(* PLC project mtcs_common, Institute of Astronomy OntoManager 0.0.1 *)
(* stored: creationDateTime 2017-02-10T20:20:17.105900, modificationDateTime 2017-02-10T20:20:17.105900 *)

TYPE InitializationStates : (SHUTDOWN := 0, INITIALIZING := 1, INITIALIZING_FAILED := 2, INITIALIZED := 3, LOCKED := 4);
END_TYPE

TYPE OperatorStates : (NONE := 0, OBSERVER := 1, TECH := 2);
END_TYPE

TYPE OperatingStates : (AUTO := 0, MANUAL := 1);
END_TYPE

TYPE LimitSwitches : (POSITIVE_LIMIT_SWITCH := 0, NEGATIVE_LIMIT_SWITCH := 1);
END_TYPE

TYPE Units : (DEGREE := 0, RADIAN := 1, PERCENT := 2, RADIANS_PER_SECOND := 3, DEGREES_PER_SECOND := 4, MILLIMETERS_PER_SECOND := 5, REVOLUTIONS_PER_SECOND := 6, REVOLUTIONS_PER_MINUTE := 7, AMPS := 8, MILLIAMPS := 9, MILLIMETER := 10, MICROMETER := 11, DEGREES_CELSIUS := 12, KELVIN := 13, BAR := 14, PASCAL := 15, UNITLESS := 16, NEWTON := 17, DECANEWTON := 18, VOLT := 19, MILLIVOLT := 20, HERTZ := 21, G := 22, MILLIG := 23, NEWTONMETER := 24, ARCSECONDS := 25, ARCSECONDS_PER_SECOND := 26, RADIANS_PER_SQUARE_SECOND := 27, DEGREES_PER_SQUARE_SECOND := 28, ARCSECONDS_PER_SQUARE_SECOND := 29, METERS_PER_SECOND := 30, HECTOPASCAL := 31, SECONDS := 32, MINUTES := 33, MILLIMETERS_PER_HOUR := 34, HITS_PER_SQUARE_CENTIMETER := 35, HITS_PER_SQUARE_CENTIMETER_PER_HOUR := 36);
END_TYPE

TYPE RequestResults : (ACCEPTED := 0, REJECTED := 1);
END_TYPE

TYPE DriveOperatingModes : (OPERATING_MODE_NONE := 0, OPERATING_MODE_TORQUE_CONTROL := 1, OPERATING_MODE_VELOCITY_CONTROL := 2, OPERATING_MODE_POSITION_CONTROL := 3);
END_TYPE

TYPE DriveBrakeStates : (BRAKE_AUTOMATIC := 0, BRAKE_FORCE_LOCK := 1, BRAKE_FORCE_UNLOCK := 2);
END_TYPE

TYPE AX52XXDriveParts : STRUCT
  channelA : AX52XXDriveChannel;  (* Channel A *)
  channelB : AX52XXDriveChannel;  (* Channel B *)
END_STRUCT;
END_TYPE

TYPE BaseAxisProcesses : STRUCT
  moveAbsolute : McMoveAbsoluteProcess;  (* Move absolute *)
  moveRelative : McMoveRelativeProcess;  (* Move relative *)
  moveVelocity : McMoveVelocityProcess;  (* Move at a constant velocity *)
  reset : McProcess;  (* Reset any errors *)
  stop : McProcess;  (* Stop any movement *)
  stopParametrized : McStopProcess;  (* Stop any movement *)
  power : McPowerProcess;  (* Power on/off the axis *)
  gearIn : McProcess;  (* Couple to master axis *)
  gearOut : McProcess;  (* Decouple from master axis *)
  initialize : Process;  (* Start initializing the axis *)
  setPosition : McSetPositionProcess;  (* Set the axis position *)
  enableExtSetGen : McProcess;  (* Enable the external setpoint generator *)
  disableExtSetGen : McProcess;  (* Disable the external setpoint generator *)
  forceCalibration : McProcess;  (* Force the calibration (homing) flag to TRUE *)
  resetCalibration : McProcess;  (* Reset the calibration (homing) flag to FALSE *)
  readParameter : McReadParameter;  (* Read a numerical parameter *)
  readBoolParameter : McReadBoolParameter;  (* Read a boolean parameter *)
  writeParameter : McWriteParameter;  (* Write a numerical parameter *)
  writeBoolParameter : McWriteBoolParameter;  (* Write a boolean parameter *)
END_STRUCT;
END_TYPE

TYPE FaulhaberDriveProcesses : STRUCT
  write : SDOWriteProcess;  (* Write a number of bytes to the drive *)
  read : SDOReadProcess;  (* Read a number of bytes from the drive *)
  initialize : Process;  (* Initialize the drive according to the config *)
END_STRUCT;
END_TYPE

TYPE AX52XXDriveChannelProcesses : STRUCT
  read : SoEReadProcess;  (* Read a number of bytes from the drive *)
  write : SoEWriteProcess;  (* Write a number of bytes to the drive *)
  update : Process;  (* Update the actual values *)
  reset : SoEResetProcess;  (* Reset the drive channel *)
  acknowledgeSafetyError : Process;  (* Acknowledge the safety card error state *)
  setBrake : SetBrakeProcess;  (* Update the actual values *)
END_STRUCT;
END_TYPE

TYPE IncrementalEncoderProcesses : STRUCT
  enableCounterResetC : Process;  (* Enable the counter reset on the C pulse *)
  disableCounterResetC : Process;  (* Disable the counter reset on the C pulse *)
END_STRUCT;
END_TYPE

TYPE SimpleRelayProcesses : STRUCT
  setEnabled : SetEnabledProcess;  (* Set the relay enabled or disabled *)
END_STRUCT;
END_TYPE

TYPE ConfigManagerProcesses : STRUCT
  save : WriteXmlProcess;  (* Save the currently active config to disk *)
  load : ReadXmlProcess;  (* Load the config from disk *)
  activate : ActivateProcess;  (* Activate the loaded config *)
END_STRUCT;
END_TYPE

TYPE ModbusRTUBusProcesses : STRUCT
  readCoil : ModbusRTUBusReadCoilProcess;  (* Read coil *)
  writeCoil : ModbusRTUBusWriteCoilProcess;  (* Write coil *)
  readRegister : ModbusRTUBusReadRegisterProcess;  (* Read register *)
  writeRegister : ModbusRTUBusWriteRegisterProcess;  (* Write register *)
END_STRUCT;
END_TYPE

TYPE BaseProcessStatuses : STRUCT
  enabledStatus : EnabledStatus;  (* Is the process enabled or not? *)
  busyStatus : BusyStatus;  (* Is the process busy or not? *)
  healthStatus : HealthStatus;  (* Is the process in a healthy state or not? *)
  startedStatus : StartedStatus;  (* Is the process started or not? *)
END_STRUCT;
END_TYPE

TYPE ProcessStepStatuses : STRUCT
  enabledStatus : EnabledStatus;  (* Is the process step enabled or not? *)
END_STRUCT;
END_TYPE

TYPE BaseAxisStatuses : STRUCT
  busyStatus : BusyStatus;  (* Is the NcAxis in a busy state? *)
  healthStatus : HealthStatus;  (* Is the NcAxis in a healthy state? *)
  poweredStatus : PoweredStatus;  (* Is the NcAxis powered? *)
  extSetGenStatus : EnabledStatus;  (* Is the NcAxis its external setpoint generator enabled? *)
  motionStatus : MotionStatus;  (* Is the NcAxis moving forward or backward or standing still? *)
END_STRUCT;
END_TYPE

TYPE FaulhaberDriveStatuses : STRUCT
  busyStatus : BusyStatus;  (* Is the NcAxis in a busy state? *)
  healthStatus : HealthStatus;  (* Is the NcAxis in a healthy state? *)
END_STRUCT;
END_TYPE

TYPE AX52XXDriveChannelStatuses : STRUCT
  busyStatus : BusyStatus;  (* Is the drive in a busy state? *)
  healthStatus : HealthStatus;  (* Is the drive in a healthy state? *)
END_STRUCT;
END_TYPE

TYPE AX52XXDriveStatuses : STRUCT
  busyStatus : BusyStatus;  (* Is the drive in a busy state? *)
  healthStatus : HealthStatus;  (* Is the drive in a healthy state? *)
END_STRUCT;
END_TYPE

TYPE SSIEncoderStatuses : STRUCT
  healthStatus : HealthStatus;  (* Is the device in a healthy state? *)
END_STRUCT;
END_TYPE

TYPE IncrementalEncoderStatuses : STRUCT
  healthStatus : HealthStatus;  (* Is the device in a healthy state? *)
  busyStatus : BusyStatus;  (* Is the device in a busy state? *)
END_STRUCT;
END_TYPE

TYPE EtherCatDeviceStatuses : STRUCT
  healthStatus : HealthStatus;  (* Is the device in a healthy state? *)
END_STRUCT;
END_TYPE

TYPE CANopenBusStatuses : STRUCT
  healthStatus : HealthStatus;  (* Is the device in a healthy state? *)
END_STRUCT;
END_TYPE

TYPE CurrentMeasurementStatuses : STRUCT
  healthStatus : HealthStatus;  (* Is the measurement valid? *)
END_STRUCT;
END_TYPE

TYPE VoltageMeasurementStatuses : STRUCT
  enabledStatus : EnabledStatus;  (* Is the voltage being measured? *)
  healthStatus : HealthStatus;  (* Is the measurement OK? *)
  alarmStatus : HiHiLoLoAlarmStatus;  (* Alarm status *)
END_STRUCT;
END_TYPE

TYPE TemperatureMeasurementStatuses : STRUCT
  enabledStatus : EnabledStatus;  (* Is the temperature being measured? *)
  healthStatus : HealthStatus;  (* Is the measurement OK? *)
  alarmStatus : HiHiLoLoAlarmStatus;  (* Alarm status *)
END_STRUCT;
END_TYPE

TYPE PressureMeasurementStatuses : STRUCT
  enabledStatus : EnabledStatus;  (* Is the pressure being measured? *)
  healthStatus : HealthStatus;  (* Is the measurement OK? *)
  alarmStatus : HiHiLoLoAlarmStatus;  (* Alarm status *)
END_STRUCT;
END_TYPE

TYPE FrequencyMeasurementStatuses : STRUCT
  enabledStatus : EnabledStatus;  (* Is the frequency being measured? *)
  healthStatus : HealthStatus;  (* Is the measurement OK? *)
  alarmStatus : HiHiLoLoAlarmStatus;  (* Alarm status *)
END_STRUCT;
END_TYPE

TYPE GForceMeasurementStatuses : STRUCT
  healthStatus : HealthStatus;  (* Is the measurement OK? *)
END_STRUCT;
END_TYPE

TYPE RelativeHumidityMeasurementStatuses : STRUCT
  enabledStatus : EnabledStatus;  (* Is the relative humidity being measured? *)
  healthStatus : HealthStatus;  (* Is the measurement OK? *)
  alarmStatus : HiHiLoLoAlarmStatus;  (* Alarm status *)
END_STRUCT;
END_TYPE

TYPE ForceMeasurementStatuses : STRUCT
  enabledStatus : EnabledStatus;  (* Is the force being measured? *)
  healthStatus : HealthStatus;  (* Is the measurement OK? *)
  alarmStatus : HiHiLoLoAlarmStatus;  (* Alarm status *)
END_STRUCT;
END_TYPE

TYPE LinearPositionMeasurement16Statuses : STRUCT
  enabledStatus : EnabledStatus;  (* Is the position being measured? *)
  healthStatus : HealthStatus;  (* Is the measurement OK? *)
  alarmStatus : HiHiLoLoAlarmStatus;  (* Alarm status *)
END_STRUCT;
END_TYPE

TYPE LinearPositionMeasurementU32Statuses : STRUCT
  enabledStatus : EnabledStatus;  (* Is the position being measured? *)
  healthStatus : HealthStatus;  (* Is the measurement OK? *)
  alarmStatus : HiHiLoLoAlarmStatus;  (* Alarm status *)
END_STRUCT;
END_TYPE

TYPE SimpleRelayStatuses : STRUCT
  busyStatus : BusyStatus;  (* Is the SimpleRelay in a busy state? *)
END_STRUCT;
END_TYPE

TYPE ConfigManagerStatuses : STRUCT
  busyStatus : BusyStatus;  (* Is the config manager in a busy state? *)
  healthStatus : HealthStatus;  (* Is the config manager in a healthy state? *)
END_STRUCT;
END_TYPE

TYPE ModbusRTUBusStatuses : STRUCT
  busyStatus : BusyStatus;  (* Is the config manager in a busy state? *)
END_STRUCT;
END_TYPE

TYPE HiHiLoLoAlarmConfig : STRUCT
  enabled : BOOL;  (* Is the alarm enabled? *)
  loLo : LREAL;  (* LowLow alarm limit (produces ERROR) *)
  lo : LREAL;  (* Low alarm limit (produces WARNING) *)
  hi : LREAL;  (* High alarm limit (produces WARNING) *)
  hiHi : LREAL;  (* HighHigh alarm limit (produces ERROR) *)
END_STRUCT;
END_TYPE

TYPE MeasurementConfig : STRUCT
  enabled : BOOL;  (* Is the quantity being measured? (Can be false e.g. if the sensor is deliberately not connected (yet).) *)
  offset : LREAL;  (* Offset to be added to the measured value (default: 0 = no offset) *)
  alarms : HiHiLoLoAlarmConfig;  (* Config *)
END_STRUCT;
END_TYPE

TYPE FaulhaberDriveConfig : STRUCT
  sendAtInitialization : BOOL;  (* Send the complete config to the drive during initialization *)
  CANopenBusNetId : STRING;  (* The CANopen bus NetId, as configured via TwinCAT, e.g. '172.16.2.131.2.1' *)
  CANopenNodePort : UINT;  (* The CANopen node port number, as configured via TwinCAT, e.g. 1005 *)
  modesOfOperation : USINT;  (* 0x6060.0: Operating mode changeover *)
  polarity : USINT;  (* 0x607E.0: Direction of rotation *)
  maxProfileVelocity : UDINT;  (* 0x607F.0: Maximum velocity, in rpm *)
  negativeLimitSwitch : USINT;  (* 0x2310.1: Lower limit switch configuration *)
  positiveLimitSwitch : USINT;  (* 0x2310.2: Upper limit switch configuration *)
  homingSwitch : USINT;  (* 0x2310.3: Homing switch configuration *)
  limitSwitchPolarity : USINT;  (* 0x2310.5: Limit switch positive edge *)
  continuousCurrentLimit : UINT;  (* 0x2333.1: Continuous current limit, in milliamps *)
  peakCurrentLimit : UINT;  (* 0x2333.2: Peak current limit, in milliamps *)
  velocityControlProportionalTerm : UINT;  (* 0x2331.1: Proportional term (gain) of the velocity control mode *)
  velocityControlIntegralTerm : UINT;  (* 0x2331.2: Integral term (gain) of the velocity control mode *)
END_STRUCT;
END_TYPE

TYPE InstrumentConfig : STRUCT
  name : STRING;  (* Name of the instrument *)
  doInitialThermalFocus : BOOL;  (* Do a thermal focus when changing to this instrument *)
  changeM3 : BOOL;  (* Change M3 to the focal station with the same name as the instrument *)
  moveKnownPosition : BOOL;  (* Move the axes to a known position (defined by the 'moveKnownPositionName' config entry) before turning off derotators *)
  moveKnownPositionName : STRING;  (* Name of the known position to move to before turning off derotators *)
  powerOnRoc : BOOL;  (* Turn on the Cassegrain derotator if needed *)
  powerOffRoc : BOOL;  (* Turn off the Cassegrain derotator if needed *)
  powerOnRon : BOOL;  (* Turn on the Nasmyth B derotator if needed *)
  powerOffRon : BOOL;  (* Turn off the Nasmyth B derotator if needed *)
  loadPointingModel : BOOL;  (* Load the pointing model with the same name as the instrument *)
  rocActive : BOOL;  (* True if the Cassegrain rotator is active (irrespective of its power status). *)
  ronActive : BOOL;  (* True if the Nasmyth rotator is active (irrespective of its power status) *)
END_STRUCT;
END_TYPE

TYPE ChangeSetpointProcessArgs : STRUCT
  setpoint : LREAL;  (* New setpoint value *)
END_STRUCT;
END_TYPE

TYPE McMoveAbsoluteProcessArgs : STRUCT
  position : LREAL;  (* New position setpoint *)
  maxVelocity : LREAL;  (* Maximum velocity *)
END_STRUCT;
END_TYPE

TYPE McMoveRelativeProcessArgs : STRUCT
  distance : LREAL;  (* Distance to move *)
  maxVelocity : LREAL;  (* Maximum velocity *)
END_STRUCT;
END_TYPE

TYPE McPowerProcessArgs : STRUCT
  enable : BOOL;  (* Enable the power or not *)
END_STRUCT;
END_TYPE

TYPE McSetPositionProcessArgs : STRUCT
  value : LREAL;  (* New position to be taken over by the encoder *)
END_STRUCT;
END_TYPE

TYPE McStopProcessArgs : STRUCT
  deceleration : LREAL;  (* Deceleration (use 0 for default). If non zero, then also jerk must be non zero! *)
  jerk : LREAL;  (* Jerk (use 0 for default). If non zero, then also deceleration must be non zero! *)
END_STRUCT;
END_TYPE

TYPE McMoveVelocityProcessArgs : STRUCT
  value : LREAL;  (* New velocity *)
END_STRUCT;
END_TYPE

TYPE SetEnabledProcessArgs : STRUCT
  enabled : BOOL;  (* True to enable, false to disable *)
END_STRUCT;
END_TYPE

TYPE McWriteParameterArgs : STRUCT
  parameterNumber : INT;  (* Number of the parameter *)
  value : LREAL;  (* Value to write *)
END_STRUCT;
END_TYPE

TYPE McReadParameterArgs : STRUCT
  parameterNumber : INT;  (* Number of the parameter *)
END_STRUCT;
END_TYPE

TYPE McWriteBoolParameterArgs : STRUCT
  parameterNumber : INT;  (* Number of the parameter *)
  value : BOOL;  (* Value to write *)
END_STRUCT;
END_TYPE

TYPE McReadBoolParameterArgs : STRUCT
  parameterNumber : INT;  (* Number of the parameter *)
END_STRUCT;
END_TYPE

TYPE SDOReadProcessArgs : STRUCT
  index : UINT;  (* SDO Index *)
  subindex : USINT;  (* SDO SubIndex *)
  noOfBytes : UDINT;  (* Number of bytes to be read *)
END_STRUCT;
END_TYPE

TYPE SDOWriteProcessArgs : STRUCT
  index : UINT;  (* SDO Index *)
  subindex : USINT;  (* SDO SubIndex *)
  noOfBytes : UDINT;  (* Number of bytes to be written *)
  value1Byte : USINT;  (* Value to be written if noOfBytes is 1 *)
  value2Bytes : UINT;  (* Value to be written if noOfBytes is 2 *)
  value4Bytes : UDINT;  (* Value to be written if noOfBytes is 4 *)
END_STRUCT;
END_TYPE

TYPE SoEReadProcessArgs : STRUCT
  index : UINT;  (* SDO Index *)
  noOfBytes : UDINT;  (* Number of bytes to be read *)
END_STRUCT;
END_TYPE

TYPE SoEWriteProcessArgs : STRUCT
  index : UINT;  (* SDO Index *)
  noOfBytes : UDINT;  (* Number of bytes to be written *)
  value1Byte : USINT;  (* Value to be written if noOfBytes is 1 *)
  value2Bytes : UINT;  (* Value to be written if noOfBytes is 2 *)
  value4Bytes : UDINT;  (* Value to be written if noOfBytes is 4 *)
END_STRUCT;
END_TYPE

TYPE SetBrakeProcessArgs : STRUCT
  newState : DriveBrakeStates;  (* Requested brake state *)
END_STRUCT;
END_TYPE

TYPE ChangeOperatingStateProcessArgs : STRUCT
  state : OperatingStates;  (* New operating state (e.g. AUTO, MANUAL) *)
END_STRUCT;
END_TYPE

TYPE ChangeOperatorStateProcessArgs : STRUCT
  state : OperatorStates;  (* New operator state (e.g. OBSERVER, TECH, ...) *)
  password : STRING;  (* Password (only sometimes required, e.g. to go from OBSERVER to TECH) *)
END_STRUCT;
END_TYPE

TYPE ReadXmlProcessArgs : STRUCT
  filePath : STRING;  (* Full path of the filename to read *)
END_STRUCT;
END_TYPE

TYPE WriteXmlProcessArgs : STRUCT
  filePath : STRING;  (* Full path of the filename to write *)
END_STRUCT;
END_TYPE

TYPE ModbusRTUBusReadCoilProcessArgs : STRUCT
  unitID : USINT;  (* Modbus station address (1..247) *)
  address : UINT;  (* Modbus data address *)
END_STRUCT;
END_TYPE

TYPE ModbusRTUBusWriteCoilProcessArgs : STRUCT
  unitID : USINT;  (* Modbus station address (1..247) *)
  address : UINT;  (* Modbus data address *)
  value : BOOL;  (* Value to write on the coil *)
END_STRUCT;
END_TYPE

TYPE ModbusRTUBusReadRegisterProcessArgs : STRUCT
  unitID : USINT;  (* Modbus station address (1..247) *)
  address : UINT;  (* Modbus data address *)
END_STRUCT;
END_TYPE

TYPE ModbusRTUBusWriteRegisterProcessArgs : STRUCT
  unitID : USINT;  (* Modbus station address (1..247) *)
  address : UINT;  (* Modbus data address *)
  value : INT;  (* Value to write on the register *)
END_STRUCT;
END_TYPE

FUNCTION_BLOCK ApertureStatus
  VAR_INPUT
    superState : BOOL := TRUE;  (* Super state (TRUE if the super state is active, or if there is no super state) *)
    isOpen : BOOL;  (* TRUE if the 'open' limit switch is active *)
    isClosed : BOOL;  (* TRUE if the 'open' limit switch is active *)
  END_VAR
  VAR_OUTPUT
    {attribute 'OPC.UA.DA' := '1'}
    {attribute 'OPC.UA.DA.Access' := '1'}
    open : BOOL;  (* The aperture is open *)
    {attribute 'OPC.UA.DA' := '1'}
    {attribute 'OPC.UA.DA.Access' := '1'}
    closed : BOOL;  (* The aperture is closed *)
    {attribute 'OPC.UA.DA' := '1'}
    {attribute 'OPC.UA.DA.Access' := '1'}
    partiallyOpen : BOOL;  (* The aperture is partially open *)
    {attribute 'OPC.UA.DA' := '1'}
    {attribute 'OPC.UA.DA.Access' := '1'}
    undefined : BOOL;  (* The aperture status is undefined *)
  END_VAR

            undefined := (isOpen AND isClosed) AND superState;
open := (isOpen AND (NOT(isClosed))) AND superState;
closed := (isClosed AND (NOT(isOpen))) AND superState;
partiallyOpen := (NOT(isOpen OR isClosed)) AND superState;

          
END_FUNCTION_BLOCK

FUNCTION_BLOCK BusyStatus
  VAR_INPUT
    superState : BOOL := TRUE;  (* Super state (TRUE if the super state is active, or if there is no super state) *)
    isBusy : BOOL;  (* TRUE if busy *)
  END_VAR
  VAR_OUTPUT
    {attribute 'OPC.UA.DA' := '1'}
    {attribute 'OPC.UA.DA.Access' := '1'}
    idle : BOOL;  (* The subject is idle *)
    {attribute 'OPC.UA.DA' := '1'}
    {attribute 'OPC.UA.DA.Access' := '1'}
    busy : BOOL;  (* The subject is busy *)
  END_VAR

            busy := isBusy AND superState;
idle := (NOT(isBusy)) AND superState;

          
END_FUNCTION_BLOCK

FUNCTION_BLOCK StartedStatus
  VAR_INPUT
    superState : BOOL := TRUE;  (* Super state (TRUE if the super state is active, or if there is no super state) *)
    isStarted : BOOL;  (* TRUE if started *)
  END_VAR
  VAR_OUTPUT
    {attribute 'OPC.UA.DA' := '1'}
    {attribute 'OPC.UA.DA.Access' := '1'}
    started : BOOL;  (* The subject is started *)
    {attribute 'OPC.UA.DA' := '1'}
    {attribute 'OPC.UA.DA.Access' := '1'}
    notStarted : BOOL;  (* The subject is started *)
  END_VAR

            started := isStarted AND superState;
notStarted := (NOT(isStarted)) AND superState;

          
END_FUNCTION_BLOCK

FUNCTION_BLOCK EnabledStatus
  VAR_INPUT
    superState : BOOL := TRUE;  (* Super state (TRUE if the super state is active, or if there is no super state) *)
    isEnabled : BOOL;  (* TRUE if enabled *)
  END_VAR
  VAR_OUTPUT
    {attribute 'OPC.UA.DA' := '1'}
    {attribute 'OPC.UA.DA.Access' := '1'}
    enabled : BOOL;  (* The subject is enabled *)
    {attribute 'OPC.UA.DA' := '1'}
    {attribute 'OPC.UA.DA.Access' := '1'}
    disabled : BOOL;  (* The subject is disabled *)
  END_VAR

            disabled := (NOT(isEnabled)) AND superState;
enabled := isEnabled AND superState;

          
END_FUNCTION_BLOCK

FUNCTION_BLOCK PoweredStatus
  VAR_INPUT
    superState : BOOL := TRUE;  (* Super state (TRUE if the super state is active, or if there is no super state) *)
    isEnabled : BOOL;  (* TRUE if power is enabled *)
  END_VAR
  VAR_OUTPUT
    {attribute 'OPC.UA.DA' := '1'}
    {attribute 'OPC.UA.DA.Access' := '1'}
    enabled : BOOL;  (* The power is enabled *)
    {attribute 'OPC.UA.DA' := '1'}
    {attribute 'OPC.UA.DA.Access' := '1'}
    disabled : BOOL;  (* The power is disabled *)
  END_VAR

            disabled := (NOT(isEnabled)) AND superState;
enabled := isEnabled AND superState;

          
END_FUNCTION_BLOCK

FUNCTION_BLOCK HealthStatus
  VAR_INPUT
    superState : BOOL := TRUE;  (* Super state (TRUE if the super state is active, or if there is no super state) *)
    isGood : BOOL;  (* TRUE if the subject is in Good health *)
    hasWarning : BOOL := FALSE;  (* TRUE to add a warning to the Good health state *)
  END_VAR
  VAR_OUTPUT
    {attribute 'OPC.UA.DA' := '1'}
    {attribute 'OPC.UA.DA.Access' := '1'}
    good : BOOL;  (* The subject is in Good health *)
    {attribute 'OPC.UA.DA' := '1'}
    {attribute 'OPC.UA.DA.Access' := '1'}
    warning : BOOL;  (* The subject is in Good health, but there are one or more warnings present *)
    {attribute 'OPC.UA.DA' := '1'}
    {attribute 'OPC.UA.DA.Access' := '1'}
    bad : BOOL;  (* The subject is in Bad health *)
  END_VAR

            good := (isGood AND (NOT(hasWarning))) AND superState;
bad := (NOT(isGood)) AND superState;
warning := (isGood AND hasWarning) AND superState;

          
END_FUNCTION_BLOCK

FUNCTION_BLOCK InitializationStatus
  VAR_INPUT
    superState : BOOL := TRUE;  (* Super state (TRUE if the super state is active, or if there is no super state) *)
    state : InitializationStates;  (* Enum! *)
  END_VAR
  VAR_OUTPUT
    {attribute 'OPC.UA.DA' := '1'}
    {attribute 'OPC.UA.DA.Access' := '1'}
    shutdown : BOOL;  (* Shutdown *)
    {attribute 'OPC.UA.DA' := '1'}
    {attribute 'OPC.UA.DA.Access' := '1'}
    initializing : BOOL;  (* Initializing *)
    {attribute 'OPC.UA.DA' := '1'}
    {attribute 'OPC.UA.DA.Access' := '1'}
    initializingFailed : BOOL;  (* Initializing failed *)
    {attribute 'OPC.UA.DA' := '1'}
    {attribute 'OPC.UA.DA.Access' := '1'}
    initialized : BOOL;  (* Initialized *)
    {attribute 'OPC.UA.DA' := '1'}
    {attribute 'OPC.UA.DA.Access' := '1'}
    locked : BOOL;  (* Locked *)
  END_VAR

            initialized := (state = InitializationStates.INITIALIZED) AND superState;
locked := (state = InitializationStates.LOCKED) AND superState;
initializing := (state = InitializationStates.INITIALIZING) AND superState;
shutdown := (state = InitializationStates.SHUTDOWN) AND superState;
initializingFailed := (state = InitializationStates.INITIALIZING_FAILED) AND superState;

          
END_FUNCTION_BLOCK

FUNCTION_BLOCK MotionStatus
  VAR_INPUT
    superState : BOOL := TRUE;  (* Super state (TRUE if the super state is active, or if there is no super state) *)
    actVel : LREAL;  (* Actual velocity *)
    tolerance : LREAL;  (* Tolerance (should be positive)! *)
  END_VAR
  VAR_OUTPUT
    {attribute 'OPC.UA.DA' := '1'}
    {attribute 'OPC.UA.DA.Access' := '1'}
    forward : BOOL;  (* Moving forwared *)
    {attribute 'OPC.UA.DA' := '1'}
    {attribute 'OPC.UA.DA.Access' := '1'}
    backward : BOOL;  (* Moving backward *)
    {attribute 'OPC.UA.DA' := '1'}
    {attribute 'OPC.UA.DA.Access' := '1'}
    standstill : BOOL;  (* Standing still *)
  END_VAR

            backward := (actVel < (-(ABS(tolerance)))) AND superState;
forward := (actVel > (ABS(tolerance))) AND superState;
standstill := (NOT(forward OR backward)) AND superState;

          
END_FUNCTION_BLOCK

FUNCTION_BLOCK HiHiLoLoAlarmStatus
  VAR_INPUT
    superState : BOOL := TRUE;  (* Super state (TRUE if the super state is active, or if there is no super state) *)
    config : HiHiLoLoAlarmConfig;  (* Config *)
    value : LREAL;  (* Value in the correct units to compare to the values from the config *)
  END_VAR
  VAR_OUTPUT
    {attribute 'OPC.UA.DA' := '1'}
    {attribute 'OPC.UA.DA.Access' := '1'}
    disabled : BOOL;  (* The alarm is disabled *)
    {attribute 'OPC.UA.DA' := '1'}
    {attribute 'OPC.UA.DA.Access' := '1'}
    hiHi : BOOL;  (* HighHigh limit active *)
    {attribute 'OPC.UA.DA' := '1'}
    {attribute 'OPC.UA.DA.Access' := '1'}
    hi : BOOL;  (* High limit active *)
    {attribute 'OPC.UA.DA' := '1'}
    {attribute 'OPC.UA.DA.Access' := '1'}
    ok : BOOL;  (* The value is within normal range *)
    {attribute 'OPC.UA.DA' := '1'}
    {attribute 'OPC.UA.DA.Access' := '1'}
    lo : BOOL;  (* Low limit active *)
    {attribute 'OPC.UA.DA' := '1'}
    {attribute 'OPC.UA.DA.Access' := '1'}
    loLo : BOOL;  (* LowLow limit active *)
  END_VAR

            lo := (config.enabled AND ((value <= config.lo) AND (value < config.loLo))) AND superState;
loLo := (config.enabled AND (value <= config.loLo)) AND superState;
disabled := (NOT(config.enabled)) AND superState;
ok := (config.enabled AND ((value > config.lo) AND (value < config.hi))) AND superState;
hi := (config.enabled AND ((value >= config.hi) AND (value < config.hiHi))) AND superState;
hiHi := (config.enabled AND (value >= config.hiHi)) AND superState;

          
END_FUNCTION_BLOCK

FUNCTION_BLOCK OpeningStatus
  VAR_INPUT
    superState : BOOL := TRUE;  (* Super state (TRUE if the super state is active, or if there is no super state) *)
    isOpening : BOOL;  (* TRUE if opening *)
    isClosing : BOOL;  (* TRUE if closing *)
  END_VAR
  VAR_OUTPUT
    {attribute 'OPC.UA.DA' := '1'}
    {attribute 'OPC.UA.DA.Access' := '1'}
    opening : BOOL;  (* Opening *)
    {attribute 'OPC.UA.DA' := '1'}
    {attribute 'OPC.UA.DA.Access' := '1'}
    closing : BOOL;  (* Closing *)
    {attribute 'OPC.UA.DA' := '1'}
    {attribute 'OPC.UA.DA.Access' := '1'}
    standstill : BOOL;  (* Standing still *)
  END_VAR

            opening := (isOpening AND (NOT(isClosing))) AND superState;
standstill := (NOT(isClosing OR isOpening)) AND superState;
closing := (isClosing AND (NOT(isOpening))) AND superState;

          
END_FUNCTION_BLOCK

FUNCTION_BLOCK OperatorStatus
  VAR_INPUT
    superState : BOOL := TRUE;  (* Super state (TRUE if the super state is active, or if there is no super state) *)
    state : OperatorStates;  (* Enum! *)
  END_VAR
  VAR_OUTPUT
    {attribute 'OPC.UA.DA' := '1'}
    {attribute 'OPC.UA.DA.Access' := '1'}
    none : BOOL;  (* None *)
    {attribute 'OPC.UA.DA' := '1'}
    {attribute 'OPC.UA.DA.Access' := '1'}
    tech : BOOL;  (* Tech *)
    {attribute 'OPC.UA.DA' := '1'}
    {attribute 'OPC.UA.DA.Access' := '1'}
    observer : BOOL;  (* Observer *)
  END_VAR

            none := (state = OperatorStates.NONE) AND superState;
tech := (state = OperatorStates.TECH) AND superState;
observer := (state = OperatorStates.OBSERVER) AND superState;

          
END_FUNCTION_BLOCK

FUNCTION_BLOCK OperatingStatus
  VAR_INPUT
    superState : BOOL := TRUE;  (* Super state (TRUE if the super state is active, or if there is no super state) *)
    state : OperatingStates;  (* Enum! *)
  END_VAR
  VAR_OUTPUT
    {attribute 'OPC.UA.DA' := '1'}
    {attribute 'OPC.UA.DA.Access' := '1'}
    auto : BOOL;  (* Auto *)
    {attribute 'OPC.UA.DA' := '1'}
    {attribute 'OPC.UA.DA.Access' := '1'}
    manual : BOOL;  (* Manual *)
  END_VAR

            manual := (state = OperatingStates.MANUAL) AND superState;
auto := (state = OperatingStates.AUTO) AND superState;

          
END_FUNCTION_BLOCK

FUNCTION_BLOCK ActivityStatus
  VAR_INPUT
    superState : BOOL := TRUE;  (* Super state (TRUE if the super state is active, or if there is no super state) *)
    isMoving : BOOL;  (* TRUE if moving *)
    isAwake : BOOL;  (* TRUE if awake *)
  END_VAR
  VAR_OUTPUT
    {attribute 'OPC.UA.DA' := '1'}
    {attribute 'OPC.UA.DA.Access' := '1'}
    moving : BOOL;  (* Opening *)
    {attribute 'OPC.UA.DA' := '1'}
    {attribute 'OPC.UA.DA.Access' := '1'}
    awake : BOOL;  (* Opening *)
    {attribute 'OPC.UA.DA' := '1'}
    {attribute 'OPC.UA.DA.Access' := '1'}
    sleeping : BOOL;  (* Opening *)
  END_VAR

            awake := (isAwake AND (NOT(isMoving))) AND superState;
sleeping := (NOT(isAwake)) AND superState;
moving := (isAwake AND isMoving) AND superState;

          
END_FUNCTION_BLOCK

FUNCTION_BLOCK SM_QuantityValue
  VAR_INPUT
    {attribute 'OPC.UA.DA' := '1'}
    {attribute 'OPC.UA.DA.Access' := '1'}
    value : LREAL;  (* Numeric value *)
    {attribute 'OPC.UA.DA' := '1'}
    {attribute 'OPC.UA.DA.Access' := '1'}
    unit : Units;  (* Unit of the numeric value *)
  END_VAR
  VAR_OUTPUT
    {attribute 'OPC.UA.DA' := '1'}
    {attribute 'OPC.UA.DA.Access' := '1'}
    actualStatus : STRING;  (* Current status description *)
    previousStatus : STRING;  (* Previous status description *)
  END_VAR

            
          

{attribute 'TcRpcEnable' := '1'}
METHOD _log : BOOL
  VAR_INPUT
    name : STRING;  (* Name of this function block instance *)
  END_VAR
  VAR_IN_OUT
    buffer : LogBuffer;  (* Buffer to write all logging to *)
  END_VAR
  VAR
    subBuffer : LogBuffer;  (* Temporary buffer to write logging by parts (sub-statemachines) to *)
  END_VAR
                  LOGGER(
    name := name,
    actualStatus := THIS^.actualStatus,
    previousStatus := THIS^.previousStatus,
    buffer := buffer,
    subBuffer := subBuffer);

                
END_METHOD
END_FUNCTION_BLOCK

FUNCTION_BLOCK SM_AngularPosition
  VAR_INPUT
    {attribute 'OPC.UA.DA' := '0'}
    newDegreesValue : LREAL;  (* New position value in degrees *)
  END_VAR
  VAR_OUTPUT
    {attribute 'OPC.UA.DA' := '1'}
    {attribute 'OPC.UA.DA.Access' := '1'}
    actualStatus : STRING;  (* Current status description *)
    previousStatus : STRING;  (* Previous status description *)
    {attribute 'OPC.UA.DA' := '1'}
    {attribute 'OPC.UA.DA.Access' := '1'}
    radians : QuantityValue;  (* Angular position in radians *)
    {attribute 'OPC.UA.DA' := '1'}
    {attribute 'OPC.UA.DA.Access' := '1'}
    degrees : QuantityValue;  (* Angular position in degrees *)
    {attribute 'OPC.UA.DA' := '1'}
    {attribute 'OPC.UA.DA.Access' := '1'}
    arcseconds : QuantityValue;  (* Angular position in arcseconds *)
  END_VAR

            radians(
    value := newDegreesValue * 0.0174532925199,
    unit := Units.RADIAN);
degrees(
    value := newDegreesValue,
    unit := Units.DEGREE);
arcseconds(
    value := newDegreesValue * 3600.0,
    unit := Units.ARCSECONDS);

          

{attribute 'TcRpcEnable' := '1'}
METHOD _log : BOOL
  VAR_INPUT
    name : STRING;  (* Name of this function block instance *)
  END_VAR
  VAR_IN_OUT
    buffer : LogBuffer;  (* Buffer to write all logging to *)
  END_VAR
  VAR
    subBuffer : LogBuffer;  (* Temporary buffer to write logging by parts (sub-statemachines) to *)
  END_VAR
                  LOGGER(
    name := name,
    actualStatus := THIS^.actualStatus,
    previousStatus := THIS^.previousStatus,
    buffer := buffer,
    subBuffer := subBuffer);

                
END_METHOD
END_FUNCTION_BLOCK

FUNCTION_BLOCK SM_LinearPosition
  VAR_INPUT
    {attribute 'OPC.UA.DA' := '0'}
    newMillimetersValue : LREAL;  (* New position value in millimeters *)
  END_VAR
  VAR_OUTPUT
    {attribute 'OPC.UA.DA' := '1'}
    {attribute 'OPC.UA.DA.Access' := '1'}
    actualStatus : STRING;  (* Current status description *)
    previousStatus : STRING;  (* Previous status description *)
    {attribute 'OPC.UA.DA' := '1'}
    {attribute 'OPC.UA.DA.Access' := '1'}
    millimeters : QuantityValue;  (* Linear position in millimeters *)
    {attribute 'OPC.UA.DA' := '1'}
    {attribute 'OPC.UA.DA.Access' := '1'}
    micrometers : QuantityValue;  (* Linear position in micrometers *)
  END_VAR

            millimeters(
    value := newMillimetersValue,
    unit := Units.MILLIMETER);
micrometers(
    value := newMillimetersValue * 1000.0,
    unit := Units.MICROMETER);

          

{attribute 'TcRpcEnable' := '1'}
METHOD _log : BOOL
  VAR_INPUT
    name : STRING;  (* Name of this function block instance *)
  END_VAR
  VAR_IN_OUT
    buffer : LogBuffer;  (* Buffer to write all logging to *)
  END_VAR
  VAR
    subBuffer : LogBuffer;  (* Temporary buffer to write logging by parts (sub-statemachines) to *)
  END_VAR
                  LOGGER(
    name := name,
    actualStatus := THIS^.actualStatus,
    previousStatus := THIS^.previousStatus,
    buffer := buffer,
    subBuffer := subBuffer);

                
END_METHOD
END_FUNCTION_BLOCK

FUNCTION_BLOCK SM_AngularVelocity
  VAR_INPUT
    {attribute 'OPC.UA.DA' := '0'}
    newDegreesPerSecondValue : LREAL;  (* New velocity value in degrees per second *)
  END_VAR
  VAR_OUTPUT
    {attribute 'OPC.UA.DA' := '1'}
    {attribute 'OPC.UA.DA.Access' := '1'}
    actualStatus : STRING;  (* Current status description *)
    previousStatus : STRING;  (* Previous status description *)
    {attribute 'OPC.UA.DA' := '1'}
    {attribute 'OPC.UA.DA.Access' := '1'}
    radiansPerSecond : QuantityValue;  (* Angular velocity in radians per second *)
    {attribute 'OPC.UA.DA' := '1'}
    {attribute 'OPC.UA.DA.Access' := '1'}
    degreesPerSecond : QuantityValue;  (* Angular velocity in degrees per second *)
    {attribute 'OPC.UA.DA' := '1'}
    {attribute 'OPC.UA.DA.Access' := '1'}
    arcsecondsPerSecond : QuantityValue;  (* Angular velocity in arcseconds per second *)
  END_VAR

            radiansPerSecond(
    value := newDegreesPerSecondValue * 0.0174532925199,
    unit := Units.RADIANS_PER_SECOND);
degreesPerSecond(
    value := newDegreesPerSecondValue,
    unit := Units.DEGREES_PER_SECOND);
arcsecondsPerSecond(
    value := newDegreesPerSecondValue * 3600.0,
    unit := Units.ARCSECONDS_PER_SECOND);

          

{attribute 'TcRpcEnable' := '1'}
METHOD _log : BOOL
  VAR_INPUT
    name : STRING;  (* Name of this function block instance *)
  END_VAR
  VAR_IN_OUT
    buffer : LogBuffer;  (* Buffer to write all logging to *)
  END_VAR
  VAR
    subBuffer : LogBuffer;  (* Temporary buffer to write logging by parts (sub-statemachines) to *)
  END_VAR
                  LOGGER(
    name := name,
    actualStatus := THIS^.actualStatus,
    previousStatus := THIS^.previousStatus,
    buffer := buffer,
    subBuffer := subBuffer);

                
END_METHOD
END_FUNCTION_BLOCK

FUNCTION_BLOCK SM_AngularAcceleration
  VAR_INPUT
    {attribute 'OPC.UA.DA' := '0'}
    newDegreesPerSquareSecondValue : LREAL;  (* New velocity value in degrees per second^2 *)
  END_VAR
  VAR_OUTPUT
    {attribute 'OPC.UA.DA' := '1'}
    {attribute 'OPC.UA.DA.Access' := '1'}
    actualStatus : STRING;  (* Current status description *)
    previousStatus : STRING;  (* Previous status description *)
    {attribute 'OPC.UA.DA' := '1'}
    {attribute 'OPC.UA.DA.Access' := '1'}
    radiansPerSquareSecond : QuantityValue;  (* Angular velocity in radians per second^2 *)
    {attribute 'OPC.UA.DA' := '1'}
    {attribute 'OPC.UA.DA.Access' := '1'}
    degreesPerSquareSecond : QuantityValue;  (* Angular velocity in degrees per second^2 *)
    {attribute 'OPC.UA.DA' := '1'}
    {attribute 'OPC.UA.DA.Access' := '1'}
    arcsecondsPerSquareSecond : QuantityValue;  (* Angular velocity in arcseconds per second^2 *)
  END_VAR

            radiansPerSquareSecond(
    value := newDegreesPerSquareSecondValue * 0.0174532925199,
    unit := Units.RADIANS_PER_SQUARE_SECOND);
degreesPerSquareSecond(
    value := newDegreesPerSquareSecondValue,
    unit := Units.DEGREES_PER_SQUARE_SECOND);
arcsecondsPerSquareSecond(
    value := newDegreesPerSquareSecondValue * 3600.0,
    unit := Units.ARCSECONDS_PER_SQUARE_SECOND);

          

{attribute 'TcRpcEnable' := '1'}
METHOD _log : BOOL
  VAR_INPUT
    name : STRING;  (* Name of this function block instance *)
  END_VAR
  VAR_IN_OUT
    buffer : LogBuffer;  (* Buffer to write all logging to *)
  END_VAR
  VAR
    subBuffer : LogBuffer;  (* Temporary buffer to write logging by parts (sub-statemachines) to *)
  END_VAR
                  LOGGER(
    name := name,
    actualStatus := THIS^.actualStatus,
    previousStatus := THIS^.previousStatus,
    buffer := buffer,
    subBuffer := subBuffer);

                
END_METHOD
END_FUNCTION_BLOCK

FUNCTION_BLOCK SM_LinearVelocity
  VAR_INPUT
    {attribute 'OPC.UA.DA' := '0'}
    newMillimetersPerSecondValue : LREAL;  (* New velocity value in millimeters per second *)
  END_VAR
  VAR_OUTPUT
    {attribute 'OPC.UA.DA' := '1'}
    {attribute 'OPC.UA.DA.Access' := '1'}
    actualStatus : STRING;  (* Current status description *)
    previousStatus : STRING;  (* Previous status description *)
    {attribute 'OPC.UA.DA' := '1'}
    {attribute 'OPC.UA.DA.Access' := '1'}
    millimetersPerSecond : QuantityValue;  (* Linear velocity in millimeters per second *)
  END_VAR

            millimetersPerSecond(
    value := newMillimetersPerSecondValue,
    unit := Units.MILLIMETERS_PER_SECOND);

          

{attribute 'TcRpcEnable' := '1'}
METHOD _log : BOOL
  VAR_INPUT
    name : STRING;  (* Name of this function block instance *)
  END_VAR
  VAR_IN_OUT
    buffer : LogBuffer;  (* Buffer to write all logging to *)
  END_VAR
  VAR
    subBuffer : LogBuffer;  (* Temporary buffer to write logging by parts (sub-statemachines) to *)
  END_VAR
                  LOGGER(
    name := name,
    actualStatus := THIS^.actualStatus,
    previousStatus := THIS^.previousStatus,
    buffer := buffer,
    subBuffer := subBuffer);

                
END_METHOD
END_FUNCTION_BLOCK

FUNCTION_BLOCK SM_Voltage
  VAR_INPUT
    {attribute 'OPC.UA.DA' := '0'}
    newVoltValue : LREAL;  (* New voltage *)
  END_VAR
  VAR_OUTPUT
    {attribute 'OPC.UA.DA' := '1'}
    {attribute 'OPC.UA.DA.Access' := '1'}
    actualStatus : STRING;  (* Current status description *)
    previousStatus : STRING;  (* Previous status description *)
    {attribute 'OPC.UA.DA' := '1'}
    {attribute 'OPC.UA.DA.Access' := '1'}
    volt : QuantityValue;  (* Voltage in Volt *)
    {attribute 'OPC.UA.DA' := '1'}
    {attribute 'OPC.UA.DA.Access' := '1'}
    milliVolt : QuantityValue;  (* Voltage in millivolt *)
  END_VAR

            volt(
    value := newVoltValue,
    unit := Units.VOLT);
milliVolt(
    value := newVoltValue * 1000.0,
    unit := Units.MILLIVOLT);

          

{attribute 'TcRpcEnable' := '1'}
METHOD _log : BOOL
  VAR_INPUT
    name : STRING;  (* Name of this function block instance *)
  END_VAR
  VAR_IN_OUT
    buffer : LogBuffer;  (* Buffer to write all logging to *)
  END_VAR
  VAR
    subBuffer : LogBuffer;  (* Temporary buffer to write logging by parts (sub-statemachines) to *)
  END_VAR
                  LOGGER(
    name := name,
    actualStatus := THIS^.actualStatus,
    previousStatus := THIS^.previousStatus,
    buffer := buffer,
    subBuffer := subBuffer);

                
END_METHOD
END_FUNCTION_BLOCK

FUNCTION_BLOCK SM_GForce
  VAR_INPUT
    {attribute 'OPC.UA.DA' := '0'}
    newMilliGValue : LREAL;  (* New milliG value *)
  END_VAR
  VAR_OUTPUT
    {attribute 'OPC.UA.DA' := '1'}
    {attribute 'OPC.UA.DA.Access' := '1'}
    actualStatus : STRING;  (* Current status description *)
    previousStatus : STRING;  (* Previous status description *)
    {attribute 'OPC.UA.DA' := '1'}
    {attribute 'OPC.UA.DA.Access' := '1'}
    g : QuantityValue;  (* Acceleration in g units *)
    {attribute 'OPC.UA.DA' := '1'}
    {attribute 'OPC.UA.DA.Access' := '1'}
    milliG : QuantityValue;  (* Acceleration in in milli g units *)
  END_VAR

            g(
    value := newMilliGValue / 1000.0,
    unit := Units.G);
milliG(
    value := newMilliGValue,
    unit := Units.MILLIG);

          

{attribute 'TcRpcEnable' := '1'}
METHOD _log : BOOL
  VAR_INPUT
    name : STRING;  (* Name of this function block instance *)
  END_VAR
  VAR_IN_OUT
    buffer : LogBuffer;  (* Buffer to write all logging to *)
  END_VAR
  VAR
    subBuffer : LogBuffer;  (* Temporary buffer to write logging by parts (sub-statemachines) to *)
  END_VAR
                  LOGGER(
    name := name,
    actualStatus := THIS^.actualStatus,
    previousStatus := THIS^.previousStatus,
    buffer := buffer,
    subBuffer := subBuffer);

                
END_METHOD
END_FUNCTION_BLOCK

FUNCTION_BLOCK SM_Current
  VAR_INPUT
    {attribute 'OPC.UA.DA' := '0'}
    newAmpsValue : LREAL;  (* New current in amps *)
  END_VAR
  VAR_OUTPUT
    {attribute 'OPC.UA.DA' := '1'}
    {attribute 'OPC.UA.DA.Access' := '1'}
    actualStatus : STRING;  (* Current status description *)
    previousStatus : STRING;  (* Previous status description *)
    {attribute 'OPC.UA.DA' := '1'}
    {attribute 'OPC.UA.DA.Access' := '1'}
    amps : QuantityValue;  (* Current in amps *)
    {attribute 'OPC.UA.DA' := '1'}
    {attribute 'OPC.UA.DA.Access' := '1'}
    milliAmps : QuantityValue;  (* Current in milliamps *)
  END_VAR

            amps(
    value := newAmpsValue,
    unit := Units.AMPS);
milliAmps(
    value := newAmpsValue * 1000.0,
    unit := Units.MILLIAMPS);

          

{attribute 'TcRpcEnable' := '1'}
METHOD _log : BOOL
  VAR_INPUT
    name : STRING;  (* Name of this function block instance *)
  END_VAR
  VAR_IN_OUT
    buffer : LogBuffer;  (* Buffer to write all logging to *)
  END_VAR
  VAR
    subBuffer : LogBuffer;  (* Temporary buffer to write logging by parts (sub-statemachines) to *)
  END_VAR
                  LOGGER(
    name := name,
    actualStatus := THIS^.actualStatus,
    previousStatus := THIS^.previousStatus,
    buffer := buffer,
    subBuffer := subBuffer);

                
END_METHOD
END_FUNCTION_BLOCK

FUNCTION_BLOCK SM_Torque
  VAR_INPUT
    {attribute 'OPC.UA.DA' := '0'}
    newNewtonmeterValue : LREAL;  (* New torque in Nm *)
  END_VAR
  VAR_OUTPUT
    {attribute 'OPC.UA.DA' := '1'}
    {attribute 'OPC.UA.DA.Access' := '1'}
    actualStatus : STRING;  (* Current status description *)
    previousStatus : STRING;  (* Previous status description *)
    {attribute 'OPC.UA.DA' := '1'}
    {attribute 'OPC.UA.DA.Access' := '1'}
    newtonmeter : QuantityValue;  (* Torque in Nm *)
  END_VAR

            newtonmeter(
    value := newNewtonmeterValue,
    unit := Units.NEWTONMETER);

          

{attribute 'TcRpcEnable' := '1'}
METHOD _log : BOOL
  VAR_INPUT
    name : STRING;  (* Name of this function block instance *)
  END_VAR
  VAR_IN_OUT
    buffer : LogBuffer;  (* Buffer to write all logging to *)
  END_VAR
  VAR
    subBuffer : LogBuffer;  (* Temporary buffer to write logging by parts (sub-statemachines) to *)
  END_VAR
                  LOGGER(
    name := name,
    actualStatus := THIS^.actualStatus,
    previousStatus := THIS^.previousStatus,
    buffer := buffer,
    subBuffer := subBuffer);

                
END_METHOD
END_FUNCTION_BLOCK

FUNCTION_BLOCK SM_TorqueLimit
  VAR_INPUT
    {attribute 'OPC.UA.DA' := '0'}
    newFractionValue : LREAL;  (* New torque limit as a unitless fraction (between 0 and 1) *)
    {attribute 'OPC.UA.DA' := '0'}
    maxNewtonmeter : LREAL;  (* Newtonmeters corresponding to 100 percent (fraction=1) *)
  END_VAR
  VAR_OUTPUT
    {attribute 'OPC.UA.DA' := '1'}
    {attribute 'OPC.UA.DA.Access' := '1'}
    actualStatus : STRING;  (* Current status description *)
    previousStatus : STRING;  (* Previous status description *)
    {attribute 'OPC.UA.DA' := '1'}
    {attribute 'OPC.UA.DA.Access' := '1'}
    unitless : QuantityValue;  (* Torque limit as a unitless fraction *)
    {attribute 'OPC.UA.DA' := '1'}
    {attribute 'OPC.UA.DA.Access' := '1'}
    percent : QuantityValue;  (* Torque limit in percent *)
    {attribute 'OPC.UA.DA' := '1'}
    {attribute 'OPC.UA.DA.Access' := '1'}
    newtonmeter : QuantityValue;  (* Torque in Nm *)
  END_VAR

            unitless(
    value := newFractionValue,
    unit := Units.UNITLESS);
percent(
    value := newFractionValue * 100.0,
    unit := Units.PERCENT);
newtonmeter(
    value := newFractionValue * maxNewtonmeter,
    unit := Units.NEWTONMETER);

          

{attribute 'TcRpcEnable' := '1'}
METHOD _log : BOOL
  VAR_INPUT
    name : STRING;  (* Name of this function block instance *)
  END_VAR
  VAR_IN_OUT
    buffer : LogBuffer;  (* Buffer to write all logging to *)
  END_VAR
  VAR
    subBuffer : LogBuffer;  (* Temporary buffer to write logging by parts (sub-statemachines) to *)
  END_VAR
                  LOGGER(
    name := name,
    actualStatus := THIS^.actualStatus,
    previousStatus := THIS^.previousStatus,
    buffer := buffer,
    subBuffer := subBuffer);

                
END_METHOD
END_FUNCTION_BLOCK

FUNCTION_BLOCK SM_AverageCurrent EXTENDS Current

            SUPER^();

          
END_FUNCTION_BLOCK

FUNCTION_BLOCK SM_Duration
  VAR_INPUT
    {attribute 'OPC.UA.DA' := '0'}
    newSecondsValue : LREAL;  (* New duration in seconds *)
  END_VAR
  VAR_OUTPUT
    {attribute 'OPC.UA.DA' := '1'}
    {attribute 'OPC.UA.DA.Access' := '1'}
    actualStatus : STRING;  (* Current status description *)
    previousStatus : STRING;  (* Previous status description *)
    {attribute 'OPC.UA.DA' := '1'}
    {attribute 'OPC.UA.DA.Access' := '1'}
    seconds : QuantityValue;  (* Duration in seconds *)
    {attribute 'OPC.UA.DA' := '1'}
    {attribute 'OPC.UA.DA.Access' := '1'}
    minutes : QuantityValue;  (* Duration in minutes *)
  END_VAR

            seconds(
    value := newSecondsValue,
    unit := Units.SECONDS);
minutes(
    value := newSecondsValue / 60.0,
    unit := Units.MINUTES);

          

{attribute 'TcRpcEnable' := '1'}
METHOD _log : BOOL
  VAR_INPUT
    name : STRING;  (* Name of this function block instance *)
  END_VAR
  VAR_IN_OUT
    buffer : LogBuffer;  (* Buffer to write all logging to *)
  END_VAR
  VAR
    subBuffer : LogBuffer;  (* Temporary buffer to write logging by parts (sub-statemachines) to *)
  END_VAR
                  LOGGER(
    name := name,
    actualStatus := THIS^.actualStatus,
    previousStatus := THIS^.previousStatus,
    buffer := buffer,
    subBuffer := subBuffer);

                
END_METHOD
END_FUNCTION_BLOCK

FUNCTION_BLOCK SM_Temperature
  VAR_INPUT
    {attribute 'OPC.UA.DA' := '0'}
    newCelsiusValue : LREAL;  (* New temperature in degrees Celsius *)
  END_VAR
  VAR_OUTPUT
    {attribute 'OPC.UA.DA' := '1'}
    {attribute 'OPC.UA.DA.Access' := '1'}
    actualStatus : STRING;  (* Current status description *)
    previousStatus : STRING;  (* Previous status description *)
    {attribute 'OPC.UA.DA' := '1'}
    {attribute 'OPC.UA.DA.Access' := '1'}
    celsius : QuantityValue;  (* Temperature in degrees Celsius *)
    {attribute 'OPC.UA.DA' := '1'}
    {attribute 'OPC.UA.DA.Access' := '1'}
    kelvin : QuantityValue;  (* Temperature in Kelvin *)
  END_VAR

            celsius(
    value := newCelsiusValue,
    unit := Units.DEGREES_CELSIUS);
kelvin(
    value := newCelsiusValue + 273.15,
    unit := Units.KELVIN);

          

{attribute 'TcRpcEnable' := '1'}
METHOD _log : BOOL
  VAR_INPUT
    name : STRING;  (* Name of this function block instance *)
  END_VAR
  VAR_IN_OUT
    buffer : LogBuffer;  (* Buffer to write all logging to *)
  END_VAR
  VAR
    subBuffer : LogBuffer;  (* Temporary buffer to write logging by parts (sub-statemachines) to *)
  END_VAR
                  LOGGER(
    name := name,
    actualStatus := THIS^.actualStatus,
    previousStatus := THIS^.previousStatus,
    buffer := buffer,
    subBuffer := subBuffer);

                
END_METHOD
END_FUNCTION_BLOCK

FUNCTION_BLOCK SM_Pressure
  VAR_INPUT
    {attribute 'OPC.UA.DA' := '0'}
    newBarValue : LREAL;  (* New pressure in Bar *)
  END_VAR
  VAR_OUTPUT
    {attribute 'OPC.UA.DA' := '1'}
    {attribute 'OPC.UA.DA.Access' := '1'}
    actualStatus : STRING;  (* Current status description *)
    previousStatus : STRING;  (* Previous status description *)
    {attribute 'OPC.UA.DA' := '1'}
    {attribute 'OPC.UA.DA.Access' := '1'}
    bar : QuantityValue;  (* Pressure in Bar *)
    {attribute 'OPC.UA.DA' := '1'}
    {attribute 'OPC.UA.DA.Access' := '1'}
    pascal : QuantityValue;  (* Pressure in Pascal *)
    {attribute 'OPC.UA.DA' := '1'}
    {attribute 'OPC.UA.DA.Access' := '1'}
    hectoPascal : QuantityValue;  (* Pressure in HectoPascal *)
  END_VAR

            bar(
    value := newBarValue,
    unit := Units.BAR);
pascal(
    value := newBarValue * 100000.0,
    unit := Units.PASCAL);

          

{attribute 'TcRpcEnable' := '1'}
METHOD _log : BOOL
  VAR_INPUT
    name : STRING;  (* Name of this function block instance *)
  END_VAR
  VAR_IN_OUT
    buffer : LogBuffer;  (* Buffer to write all logging to *)
  END_VAR
  VAR
    subBuffer : LogBuffer;  (* Temporary buffer to write logging by parts (sub-statemachines) to *)
  END_VAR
                  LOGGER(
    name := name,
    actualStatus := THIS^.actualStatus,
    previousStatus := THIS^.previousStatus,
    buffer := buffer,
    subBuffer := subBuffer);

                
END_METHOD
END_FUNCTION_BLOCK

FUNCTION_BLOCK SM_Frequency
  VAR_INPUT
    {attribute 'OPC.UA.DA' := '0'}
    newHertzValue : LREAL;  (* New frequency in Hz *)
  END_VAR
  VAR_OUTPUT
    {attribute 'OPC.UA.DA' := '1'}
    {attribute 'OPC.UA.DA.Access' := '1'}
    actualStatus : STRING;  (* Current status description *)
    previousStatus : STRING;  (* Previous status description *)
    {attribute 'OPC.UA.DA' := '1'}
    {attribute 'OPC.UA.DA.Access' := '1'}
    hertz : QuantityValue;  (* Frequency in Hertz *)
  END_VAR

            hertz(
    value := newHertzValue,
    unit := Units.HERTZ);

          

{attribute 'TcRpcEnable' := '1'}
METHOD _log : BOOL
  VAR_INPUT
    name : STRING;  (* Name of this function block instance *)
  END_VAR
  VAR_IN_OUT
    buffer : LogBuffer;  (* Buffer to write all logging to *)
  END_VAR
  VAR
    subBuffer : LogBuffer;  (* Temporary buffer to write logging by parts (sub-statemachines) to *)
  END_VAR
                  LOGGER(
    name := name,
    actualStatus := THIS^.actualStatus,
    previousStatus := THIS^.previousStatus,
    buffer := buffer,
    subBuffer := subBuffer);

                
END_METHOD
END_FUNCTION_BLOCK

FUNCTION_BLOCK SM_Force
  VAR_INPUT
    {attribute 'OPC.UA.DA' := '0'}
    newNewtonValue : LREAL;  (* New force in Newton *)
  END_VAR
  VAR_OUTPUT
    {attribute 'OPC.UA.DA' := '1'}
    {attribute 'OPC.UA.DA.Access' := '1'}
    actualStatus : STRING;  (* Current status description *)
    previousStatus : STRING;  (* Previous status description *)
    {attribute 'OPC.UA.DA' := '1'}
    {attribute 'OPC.UA.DA.Access' := '1'}
    newton : QuantityValue;  (* Force in Newton *)
    {attribute 'OPC.UA.DA' := '1'}
    {attribute 'OPC.UA.DA.Access' := '1'}
    decaNewton : QuantityValue;  (* Force in decaNewton *)
  END_VAR

            newton(
    value := newNewtonValue,
    unit := Units.NEWTON);
decaNewton(
    value := newNewtonValue / 10.0,
    unit := Units.DECANEWTON);

          

{attribute 'TcRpcEnable' := '1'}
METHOD _log : BOOL
  VAR_INPUT
    name : STRING;  (* Name of this function block instance *)
  END_VAR
  VAR_IN_OUT
    buffer : LogBuffer;  (* Buffer to write all logging to *)
  END_VAR
  VAR
    subBuffer : LogBuffer;  (* Temporary buffer to write logging by parts (sub-statemachines) to *)
  END_VAR
                  LOGGER(
    name := name,
    actualStatus := THIS^.actualStatus,
    previousStatus := THIS^.previousStatus,
    buffer := buffer,
    subBuffer := subBuffer);

                
END_METHOD
END_FUNCTION_BLOCK

FUNCTION_BLOCK SM_Fraction
  VAR_INPUT
    {attribute 'OPC.UA.DA' := '0'}
    newFractionValue : LREAL;  (* New fraction (between 0 and 1) *)
  END_VAR
  VAR_OUTPUT
    {attribute 'OPC.UA.DA' := '1'}
    {attribute 'OPC.UA.DA.Access' := '1'}
    actualStatus : STRING;  (* Current status description *)
    previousStatus : STRING;  (* Previous status description *)
    {attribute 'OPC.UA.DA' := '1'}
    {attribute 'OPC.UA.DA.Access' := '1'}
    unitless : QuantityValue;  (* Fraction as a unitless value between 0 and 1 *)
    {attribute 'OPC.UA.DA' := '1'}
    {attribute 'OPC.UA.DA.Access' := '1'}
    percent : QuantityValue;  (* Fraction as a percentage value between 0 and 100 *)
  END_VAR

            unitless(
    value := newFractionValue,
    unit := Units.UNITLESS);
percent(
    value := newFractionValue * 100.0,
    unit := Units.PERCENT);

          

{attribute 'TcRpcEnable' := '1'}
METHOD _log : BOOL
  VAR_INPUT
    name : STRING;  (* Name of this function block instance *)
  END_VAR
  VAR_IN_OUT
    buffer : LogBuffer;  (* Buffer to write all logging to *)
  END_VAR
  VAR
    subBuffer : LogBuffer;  (* Temporary buffer to write logging by parts (sub-statemachines) to *)
  END_VAR
                  LOGGER(
    name := name,
    actualStatus := THIS^.actualStatus,
    previousStatus := THIS^.previousStatus,
    buffer := buffer,
    subBuffer := subBuffer);

                
END_METHOD
END_FUNCTION_BLOCK

FUNCTION_BLOCK SM_BaseProcess
  VAR_INPUT
    {attribute 'OPC.UA.DA' := '0'}
    isEnabled : BOOL;  (* Should the trigger be enabled? *)
  END_VAR
  VAR_OUTPUT
    {attribute 'OPC.UA.DA' := '1'}
    {attribute 'OPC.UA.DA.Access' := '1'}
    actualStatus : STRING;  (* Current status description *)
    previousStatus : STRING;  (* Previous status description *)
    statuses : BaseProcessStatuses;  (* Statuses of the state machine *)
  END_VAR
  VAR
    {attribute 'OPC.UA.DA' := '1'}
    do_request : BOOL;  (* Write TRUE to request the start of the process *)
    {attribute 'OPC.UA.DA' := '1'}
    do_request_result : RequestResults;  (* Result of the request *)
  END_VAR

            statuses.enabledStatus( isEnabled := isEnabled );
statuses.busyStatus();
statuses.healthStatus();
statuses.startedStatus();

          

{attribute 'TcRpcEnable' := '1'}
METHOD _log : BOOL
  VAR_INPUT
    name : STRING;  (* Name of this function block instance *)
  END_VAR
  VAR_IN_OUT
    buffer : LogBuffer;  (* Buffer to write all logging to *)
  END_VAR
  VAR
    subBuffer : LogBuffer;  (* Temporary buffer to write logging by parts (sub-statemachines) to *)
  END_VAR
                  LOGGER(
    name := name,
    actualStatus := THIS^.actualStatus,
    previousStatus := THIS^.previousStatus,
    buffer := buffer,
    subBuffer := subBuffer,
    pHealthStatus := ADR(THIS^.statuses.healthStatus),
    pBusyStatus := ADR(THIS^.statuses.busyStatus));

                
END_METHOD
END_FUNCTION_BLOCK

FUNCTION_BLOCK SM_BaseMcProcess EXTENDS BaseProcess
  VAR_INPUT
    {attribute 'OPC.UA.DA' := '1'}
    {attribute 'OPC.UA.DA.Access' := '1'}
    errorId : UDINT;  (* Error ID according to Beckhoff/PlcOpen Motion Control *)
  END_VAR

            SUPER^();

          
END_FUNCTION_BLOCK

FUNCTION_BLOCK SM_ProcessStep
  VAR_INPUT
    {attribute 'OPC.UA.DA' := '0'}
    isEnabled : BOOL;  (* Is the step enabled? *)
  END_VAR
  VAR_OUTPUT
    {attribute 'OPC.UA.DA' := '1'}
    {attribute 'OPC.UA.DA.Access' := '1'}
    actualStatus : STRING;  (* Current status description *)
    previousStatus : STRING;  (* Previous status description *)
    statuses : ProcessStepStatuses;  (* Statuses of the state machine *)
  END_VAR
  VAR_IN_OUT
    {attribute 'OPC.UA.DA' := '0'}
    process : BaseProcess;  (* The process corresponding to the step *)
  END_VAR

            statuses.enabledStatus( isEnabled := isEnabled );

          

{attribute 'TcRpcEnable' := '1'}
METHOD _log : BOOL
  VAR_INPUT
    name : STRING;  (* Name of this function block instance *)
  END_VAR
  VAR_IN_OUT
    buffer : LogBuffer;  (* Buffer to write all logging to *)
  END_VAR
  VAR
    subBuffer : LogBuffer;  (* Temporary buffer to write logging by parts (sub-statemachines) to *)
  END_VAR
                  LOGGER(
    name := name,
    actualStatus := THIS^.actualStatus,
    previousStatus := THIS^.previousStatus,
    buffer := buffer,
    subBuffer := subBuffer);

                
END_METHOD
END_FUNCTION_BLOCK

FUNCTION_BLOCK SM_BaseXmlDataSrvProcess EXTENDS BaseProcess
  VAR_INPUT
    {attribute 'OPC.UA.DA' := '1'}
    {attribute 'OPC.UA.DA.Access' := '1'}
    errorId : UDINT;  (* Error ID according to Beckhoff XML Data Server library *)
  END_VAR

            SUPER^();

          
END_FUNCTION_BLOCK

FUNCTION_BLOCK SM_BaseAxis
  VAR_INPUT
    {attribute 'OPC.UA.DA' := '1'}
    {attribute 'OPC.UA.DA.Access' := '1'}
    axis_ref : AXIS_REF;  (* The AXIS_REF to be linked to the NC I/O *)
    {attribute 'OPC.UA.DA' := '1'}
    {attribute 'OPC.UA.DA.Access' := '1'}
    isGearingSupported : BOOL := FALSE;  (* Is gearIn/gearOut supported? *)
    {attribute 'OPC.UA.DA' := '0'}
    isEnabled : BOOL;  (* Is control enabled? *)
    {attribute 'OPC.UA.DA' := '0'}
    standstillTolerance : LREAL;  (* Tolerance in [main units] per second: if < ABS(this value), then the axis is considered to be standing still *)
  END_VAR
  VAR_OUTPUT
    {attribute 'OPC.UA.DA' := '1'}
    {attribute 'OPC.UA.DA.Access' := '1'}
    actualStatus : STRING;  (* Current status description *)
    previousStatus : STRING;  (* Previous status description *)
    {attribute 'OPC.UA.DA' := '1'}
    {attribute 'OPC.UA.DA.Access' := '1'}
    isJogEnabled : BOOL;  (* True if jog is enabled *)
    statuses : BaseAxisStatuses;  (* Statuses of the state machine *)
    processes : BaseAxisProcesses;  (* Processes of the state machine *)
  END_VAR

            statuses.busyStatus( isBusy := processes.moveAbsolute.statuses.busyStatus.busy OR (processes.moveRelative.statuses.busyStatus.busy OR (processes.reset.statuses.busyStatus.busy OR (processes.power.statuses.busyStatus.busy OR (processes.gearIn.statuses.busyStatus.busy OR (processes.gearOut.statuses.busyStatus.busy OR (processes.initialize.statuses.busyStatus.busy OR (processes.setPosition.statuses.busyStatus.busy OR (processes.enableExtSetGen.statuses.busyStatus.busy OR (processes.disableExtSetGen.statuses.busyStatus.busy OR (processes.forceCalibration.statuses.busyStatus.busy OR (processes.resetCalibration.statuses.busyStatus.busy OR (processes.readParameter.statuses.busyStatus.busy OR (processes.readBoolParameter.statuses.busyStatus.busy OR (processes.writeParameter.statuses.busyStatus.busy OR processes.writeBoolParameter.statuses.busyStatus.busy)))))))))))))) );
statuses.healthStatus( isGood := NOT(axis_ref.Status.Error) );
statuses.poweredStatus( isEnabled := NOT(axis_ref.Status.Disabled) );
statuses.extSetGenStatus( isEnabled := axis_ref.Status.ExtSetPointGenEnabled );
statuses.motionStatus(
    actVel := axis_ref.NcToPlc.ActVelo,
    tolerance := standstillTolerance);
processes.moveAbsolute( isEnabled := isEnabled );
processes.moveRelative( isEnabled := isEnabled );
processes.moveVelocity( isEnabled := isEnabled AND processes.moveVelocity.statuses.busyStatus.idle );
processes.reset( isEnabled := isEnabled AND processes.reset.statuses.busyStatus.idle );
processes.stop( isEnabled := isEnabled AND processes.stop.statuses.busyStatus.idle );
processes.stopParametrized();
processes.power( isEnabled := isEnabled AND processes.power.statuses.busyStatus.idle );
processes.gearIn( isEnabled := isEnabled AND (processes.gearIn.statuses.busyStatus.idle AND isGearingSupported) );
processes.gearOut( isEnabled := isEnabled AND (processes.gearOut.statuses.busyStatus.idle AND isGearingSupported) );
processes.initialize( isEnabled := isEnabled AND statuses.busyStatus.idle );
processes.setPosition( isEnabled := isEnabled AND processes.setPosition.statuses.busyStatus.idle );
processes.enableExtSetGen( isEnabled := isEnabled AND processes.enableExtSetGen.statuses.busyStatus.idle );
processes.disableExtSetGen( isEnabled := isEnabled AND processes.disableExtSetGen.statuses.busyStatus.idle );
processes.forceCalibration( isEnabled := isEnabled AND statuses.busyStatus.idle );
processes.resetCalibration( isEnabled := isEnabled AND statuses.busyStatus.idle );
processes.readParameter( isEnabled := isEnabled AND statuses.busyStatus.idle );
processes.readBoolParameter( isEnabled := isEnabled AND statuses.busyStatus.idle );
processes.writeParameter( isEnabled := isEnabled AND statuses.busyStatus.idle );
processes.writeBoolParameter( isEnabled := isEnabled AND statuses.busyStatus.idle );

          

{attribute 'TcRpcEnable' := '1'}
METHOD moveAbsolute : RequestResults
  VAR_INPUT
    position : LREAL;
    maxVelocity : LREAL;
  END_VAR
                  moveAbsolute := THIS^.processes.moveAbsolute.request(
    position := position,
    maxVelocity := maxVelocity);

                
END_METHOD

{attribute 'TcRpcEnable' := '1'}
METHOD moveRelative : RequestResults
  VAR_INPUT
    distance : LREAL;
    maxVelocity : LREAL;
  END_VAR
                  moveRelative := THIS^.processes.moveRelative.request(
    distance := distance,
    maxVelocity := maxVelocity);

                
END_METHOD

{attribute 'TcRpcEnable' := '1'}
METHOD moveVelocity : RequestResults
  VAR_INPUT
    value : LREAL;
  END_VAR
                  moveVelocity := THIS^.processes.moveVelocity.request( value := value );

                
END_METHOD

{attribute 'TcRpcEnable' := '1'}
METHOD reset : RequestResults
                  reset := THIS^.processes.reset.request();

                
END_METHOD

{attribute 'TcRpcEnable' := '1'}
METHOD stop : RequestResults
                  stop := THIS^.processes.stop.request();

                
END_METHOD

{attribute 'TcRpcEnable' := '1'}
METHOD stopParametrized : RequestResults
  VAR_INPUT
    deceleration : LREAL;
    jerk : LREAL;
  END_VAR
                  stopParametrized := THIS^.processes.stopParametrized.request(
    deceleration := deceleration,
    jerk := jerk);

                
END_METHOD

{attribute 'TcRpcEnable' := '1'}
METHOD power : RequestResults
  VAR_INPUT
    enable : BOOL;
  END_VAR
                  power := THIS^.processes.power.request( enable := enable );

                
END_METHOD

{attribute 'TcRpcEnable' := '1'}
METHOD gearIn : RequestResults
                  gearIn := THIS^.processes.gearIn.request();

                
END_METHOD

{attribute 'TcRpcEnable' := '1'}
METHOD gearOut : RequestResults
                  gearOut := THIS^.processes.gearOut.request();

                
END_METHOD

{attribute 'TcRpcEnable' := '1'}
METHOD initialize : RequestResults
                  initialize := THIS^.processes.initialize.request();

                
END_METHOD

{attribute 'TcRpcEnable' := '1'}
METHOD setPosition : RequestResults
  VAR_INPUT
    value : LREAL;
  END_VAR
                  setPosition := THIS^.processes.setPosition.request( value := value );

                
END_METHOD

{attribute 'TcRpcEnable' := '1'}
METHOD enableExtSetGen : RequestResults
                  enableExtSetGen := THIS^.processes.enableExtSetGen.request();

                
END_METHOD

{attribute 'TcRpcEnable' := '1'}
METHOD disableExtSetGen : RequestResults
                  disableExtSetGen := THIS^.processes.disableExtSetGen.request();

                
END_METHOD

{attribute 'TcRpcEnable' := '1'}
METHOD forceCalibration : RequestResults
                  forceCalibration := THIS^.processes.forceCalibration.request();

                
END_METHOD

{attribute 'TcRpcEnable' := '1'}
METHOD resetCalibration : RequestResults
                  resetCalibration := THIS^.processes.resetCalibration.request();

                
END_METHOD

{attribute 'TcRpcEnable' := '1'}
METHOD readParameter : RequestResults
  VAR_INPUT
    parameterNumber : INT;
  END_VAR
                  readParameter := THIS^.processes.readParameter.request( parameterNumber := parameterNumber );

                
END_METHOD

{attribute 'TcRpcEnable' := '1'}
METHOD readBoolParameter : RequestResults
  VAR_INPUT
    parameterNumber : INT;
  END_VAR
                  readBoolParameter := THIS^.processes.readBoolParameter.request( parameterNumber := parameterNumber );

                
END_METHOD

{attribute 'TcRpcEnable' := '1'}
METHOD writeParameter : RequestResults
  VAR_INPUT
    parameterNumber : INT;
    value : LREAL;
  END_VAR
                  writeParameter := THIS^.processes.writeParameter.request(
    parameterNumber := parameterNumber,
    value := value);

                
END_METHOD

{attribute 'TcRpcEnable' := '1'}
METHOD writeBoolParameter : RequestResults
  VAR_INPUT
    parameterNumber : INT;
    value : BOOL;
  END_VAR
                  writeBoolParameter := THIS^.processes.writeBoolParameter.request(
    parameterNumber := parameterNumber,
    value := value);

                
END_METHOD

{attribute 'TcRpcEnable' := '1'}
METHOD _log : BOOL
  VAR_INPUT
    name : STRING;  (* Name of this function block instance *)
  END_VAR
  VAR_IN_OUT
    buffer : LogBuffer;  (* Buffer to write all logging to *)
  END_VAR
  VAR
    subBuffer : LogBuffer;  (* Temporary buffer to write logging by parts (sub-statemachines) to *)
  END_VAR
                  LOGGER(
    name := name,
    actualStatus := THIS^.actualStatus,
    previousStatus := THIS^.previousStatus,
    buffer := buffer,
    subBuffer := subBuffer,
    pHealthStatus := ADR(THIS^.statuses.healthStatus),
    pBusyStatus := ADR(THIS^.statuses.busyStatus));

                
END_METHOD
END_FUNCTION_BLOCK

FUNCTION_BLOCK SM_AngularAxis EXTENDS BaseAxis
  VAR_OUTPUT
    {attribute 'OPC.UA.DA' := '1'}
    {attribute 'OPC.UA.DA.Access' := '1'}
    actPos : AngularPosition;  (* Actual position of the axis *)
    {attribute 'OPC.UA.DA' := '1'}
    {attribute 'OPC.UA.DA.Access' := '1'}
    actVel : AngularVelocity;  (* Actual velocity of the axis *)
  END_VAR

            actPos( newDegreesValue := axis_ref.NcToPlc.ActPos );
actVel( newDegreesPerSecondValue := axis_ref.NcToPlc.ActVelo );
SUPER^();

          
END_FUNCTION_BLOCK

FUNCTION_BLOCK SM_LinearAxis EXTENDS BaseAxis
  VAR_OUTPUT
    {attribute 'OPC.UA.DA' := '1'}
    {attribute 'OPC.UA.DA.Access' := '1'}
    actPos : LinearPosition;  (* Actual position of the axis *)
    {attribute 'OPC.UA.DA' := '1'}
    {attribute 'OPC.UA.DA.Access' := '1'}
    actVel : LinearVelocity;  (* Actual velocity of the axis *)
  END_VAR

            actPos( newMillimetersValue := axis_ref.NcToPlc.ActPos );
actVel( newMillimetersPerSecondValue := axis_ref.NcToPlc.ActVelo );
SUPER^();

          
END_FUNCTION_BLOCK

FUNCTION_BLOCK SM_FaulhaberDrive
  VAR_INPUT
    {attribute 'OPC.UA.DA' := '1'}
    {attribute 'OPC.UA.DA.Access' := '1'}
    config : FaulhaberDriveConfig;  (* Faulhaber drive config *)
    {attribute 'OPC.UA.DA' := '0'}
    isEnabled : BOOL;  (* Is control enabled? *)
    {attribute 'OPC.UA.DA' := '0'}
    newMilliampsValue AT %I* : INT;  (* Current in milliamps, linked to PDO *)
  END_VAR
  VAR_OUTPUT
    {attribute 'OPC.UA.DA' := '1'}
    {attribute 'OPC.UA.DA.Access' := '1'}
    actualStatus : STRING;  (* Current status description *)
    previousStatus : STRING;  (* Previous status description *)
    {attribute 'OPC.UA.DA' := '1'}
    {attribute 'OPC.UA.DA.Access' := '1'}
    actualCurrent : Current;  (* Actual current *)
    {attribute 'OPC.UA.DA' := '1'}
    {attribute 'OPC.UA.DA.Access' := '1'}
    averageCurrent : AverageCurrent;  (* Average current *)
    statuses : FaulhaberDriveStatuses;  (* Statuses of the state machine *)
    processes : FaulhaberDriveProcesses;  (* Processes of the state machine *)
  END_VAR

            actualCurrent( newAmpsValue := newMilliampsValue / 1000.0 );
averageCurrent( newAmpsValue := newMilliampsValue / 1000.0 );
statuses.busyStatus( isBusy := processes.write.statuses.busyStatus.busy OR (processes.read.statuses.busyStatus.busy OR processes.initialize.statuses.busyStatus.busy) );
statuses.healthStatus( isGood := processes.write.statuses.healthStatus.good AND (processes.read.statuses.healthStatus.good AND processes.initialize.statuses.healthStatus.good) );
processes.write( isEnabled := isEnabled AND statuses.busyStatus.idle );
processes.read( isEnabled := isEnabled AND statuses.busyStatus.idle );
processes.initialize();

          

{attribute 'TcRpcEnable' := '1'}
METHOD write : RequestResults
  VAR_INPUT
    index : UINT;
    subindex : USINT;
    noOfBytes : UDINT;
    value1Byte : USINT;
    value2Bytes : UINT;
    value4Bytes : UDINT;
  END_VAR
                  write := THIS^.processes.write.request(
    index := index,
    subindex := subindex,
    noOfBytes := noOfBytes,
    value1Byte := value1Byte,
    value2Bytes := value2Bytes,
    value4Bytes := value4Bytes);

                
END_METHOD

{attribute 'TcRpcEnable' := '1'}
METHOD read : RequestResults
  VAR_INPUT
    index : UINT;
    subindex : USINT;
    noOfBytes : UDINT;
  END_VAR
                  read := THIS^.processes.read.request(
    index := index,
    subindex := subindex,
    noOfBytes := noOfBytes);

                
END_METHOD

{attribute 'TcRpcEnable' := '1'}
METHOD initialize : RequestResults
                  initialize := THIS^.processes.initialize.request();

                
END_METHOD

{attribute 'TcRpcEnable' := '1'}
METHOD _log : BOOL
  VAR_INPUT
    name : STRING;  (* Name of this function block instance *)
  END_VAR
  VAR_IN_OUT
    buffer : LogBuffer;  (* Buffer to write all logging to *)
  END_VAR
  VAR
    subBuffer : LogBuffer;  (* Temporary buffer to write logging by parts (sub-statemachines) to *)
  END_VAR
                  LOGGER(
    name := name,
    actualStatus := THIS^.actualStatus,
    previousStatus := THIS^.previousStatus,
    buffer := buffer,
    subBuffer := subBuffer,
    pHealthStatus := ADR(THIS^.statuses.healthStatus),
    pBusyStatus := ADR(THIS^.statuses.busyStatus));

                
END_METHOD
END_FUNCTION_BLOCK

FUNCTION_BLOCK SM_AX52XXDriveChannel
  VAR_INPUT
    {attribute 'OPC.UA.DA' := '1'}
    {attribute 'OPC.UA.DA.Access' := '1'}
    errorC1D AT %I* : INT;  (* Class 1 Diagnostic (C1D *)
    {attribute 'OPC.UA.DA' := '1'}
    {attribute 'OPC.UA.DA.Access' := '1'}
    isEnabled : BOOL;  (* Is control enabled? *)
    {attribute 'OPC.UA.DA' := '1'}
    {attribute 'OPC.UA.DA.Access' := '1'}
    torqueFeedbackValue AT %I* : INT;  (* Torque feedback, cyclically updated by the drive channel *)
    {attribute 'OPC.UA.DA' := '1'}
    {attribute 'OPC.UA.DA.Access' := '1'}
    torqueCommandValue AT %Q* : INT;  (* Torque command (only in case of torque control!) *)
    {attribute 'OPC.UA.DA' := '1'}
    {attribute 'OPC.UA.DA.Access' := '1'}
    digitalInputs AT %I* : INT;  (* Digital inputs (e.g. bit 0 = 1 if input 0 = high), cyclically updated by the drive channel *)
    {attribute 'OPC.UA.DA' := '1'}
    {attribute 'OPC.UA.DA.Access' := '1'}
    digitalOutputs AT %Q* : INT;  (* Digital outputs (e.g. bit 0 = 1 if input 0 = high), cyclically updated by the drive channel *)
    {attribute 'OPC.UA.DA' := '1'}
    {attribute 'OPC.UA.DA.Access' := '1'}
    safetyOptionState AT %I* : INT;  (* Safety option state (P-0-2002) *)
    {attribute 'OPC.UA.DA' := '1'}
    {attribute 'OPC.UA.DA.Access' := '1'}
    diagnosticNumber AT %I* : UDINT;  (* Diagnostic number *)
  END_VAR
  VAR_OUTPUT
    {attribute 'OPC.UA.DA' := '1'}
    {attribute 'OPC.UA.DA.Access' := '1'}
    actualStatus : STRING;  (* Current status description *)
    previousStatus : STRING;  (* Previous status description *)
    {attribute 'OPC.UA.DA' := '1'}
    {attribute 'OPC.UA.DA.Access' := '1'}
    isInSafetate : BOOL;  (* True if the drive is in safe state *)
    {attribute 'OPC.UA.DA' := '1'}
    {attribute 'OPC.UA.DA.Access' := '1'}
    actualTorqueFeedback : Torque;  (* The actual torque feedback value (updated constantly!) *)
    {attribute 'OPC.UA.DA' := '1'}
    {attribute 'OPC.UA.DA.Access' := '1'}
    channelPeakCurrent : Current;  (* The configured channel peak current *)
    {attribute 'OPC.UA.DA' := '1'}
    {attribute 'OPC.UA.DA.Access' := '1'}
    channelRatedCurrent : Current;  (* The configured channel peak current *)
    {attribute 'OPC.UA.DA' := '1'}
    {attribute 'OPC.UA.DA.Access' := '1'}
    continuousStallTorque : Torque;  (* The motor continuous stall torque *)
    {attribute 'OPC.UA.DA' := '1'}
    {attribute 'OPC.UA.DA.Access' := '1'}
    continuousStallCurrent : Current;  (* The motor continuous stall current *)
    {attribute 'OPC.UA.DA' := '1'}
    {attribute 'OPC.UA.DA.Access' := '1'}
    torqueConstant : LREAL;  (* The motor torque constant, in Nm/A *)
    {attribute 'OPC.UA.DA' := '1'}
    {attribute 'OPC.UA.DA.Access' := '1'}
    bipolarTorqueLimit : TorqueLimit;  (* The drive bipolar torque limit *)
    {attribute 'OPC.UA.DA' := '1'}
    {attribute 'OPC.UA.DA.Access' := '1'}
    positiveTorqueLimit : TorqueLimit;  (* The drive positive torque limit *)
    {attribute 'OPC.UA.DA' := '1'}
    {attribute 'OPC.UA.DA.Access' := '1'}
    negativeTorqueLimit : TorqueLimit;  (* The drive negative torque limit *)
    {attribute 'OPC.UA.DA' := '1'}
    {attribute 'OPC.UA.DA.Access' := '1'}
    operatingMode : DriveOperatingModes;  (* The drive operating mode, as an ENUM value *)
    {attribute 'OPC.UA.DA' := '1'}
    {attribute 'OPC.UA.DA.Access' := '1'}
    operatingModeDescription : STRING;  (* The drive operating mode, as a descriptive text *)
    {attribute 'OPC.UA.DA' := '1'}
    {attribute 'OPC.UA.DA.Access' := '1'}
    brakeState : DriveBrakeStates;  (* The drive brake state, as an ENUM value *)
    {attribute 'OPC.UA.DA' := '1'}
    {attribute 'OPC.UA.DA.Access' := '1'}
    brakeStateDescription : STRING;  (* The drive brake state, as a descriptive text *)
    {attribute 'OPC.UA.DA' := '1'}
    {attribute 'OPC.UA.DA.Access' := '1'}
    torqueCommand : TorqueLimit;  (* The torque command (only in case of torque control!) *)
    {attribute 'OPC.UA.DA' := '1'}
    {attribute 'OPC.UA.DA.Access' := '1'}
    safetyErrorAck AT %Q* : BOOL;  (* Error acknowledge of AX5805 safety card *)
    statuses : AX52XXDriveChannelStatuses;  (* Statuses of the state machine *)
    processes : AX52XXDriveChannelProcesses;  (* Processes of the state machine *)
  END_VAR

            actualTorqueFeedback( newNewtonmeterValue := ((torqueFeedbackValue / 1000.0) * channelPeakCurrent.amps.value) * torqueConstant );
torqueCommand(
    newFractionValue := torqueCommandValue / 1000.0,
    maxNewtonmeter := channelPeakCurrent.amps.value * torqueConstant);
statuses.busyStatus( isBusy := processes.write.statuses.busyStatus.busy OR (processes.read.statuses.busyStatus.busy OR (processes.update.statuses.busyStatus.busy OR (processes.reset.statuses.busyStatus.busy OR processes.acknowledgeSafetyError.statuses.busyStatus.busy))) );
statuses.healthStatus(
    isGood := processes.write.statuses.healthStatus.isGood AND (processes.read.statuses.healthStatus.isGood AND (processes.update.statuses.healthStatus.isGood AND (processes.reset.statuses.healthStatus.isGood AND processes.acknowledgeSafetyError.statuses.healthStatus.isGood))),
    hasWarning := processes.write.statuses.healthStatus.hasWarning OR (processes.read.statuses.healthStatus.hasWarning OR (processes.update.statuses.healthStatus.hasWarning OR (processes.reset.statuses.healthStatus.hasWarning OR processes.acknowledgeSafetyError.statuses.healthStatus.hasWarning))));
processes.read( isEnabled := isEnabled AND statuses.busyStatus.idle );
processes.write( isEnabled := isEnabled AND statuses.busyStatus.idle );
processes.update( isEnabled := statuses.busyStatus.idle );
processes.reset( isEnabled := statuses.busyStatus.idle );
processes.acknowledgeSafetyError( isEnabled := isEnabled AND processes.acknowledgeSafetyError.statuses.busyStatus.idle );
processes.setBrake( isEnabled := isEnabled AND statuses.busyStatus.idle );

          

{attribute 'TcRpcEnable' := '1'}
METHOD read : RequestResults
  VAR_INPUT
    index : UINT;
    noOfBytes : UDINT;
  END_VAR
                  read := THIS^.processes.read.request(
    index := index,
    noOfBytes := noOfBytes);

                
END_METHOD

{attribute 'TcRpcEnable' := '1'}
METHOD write : RequestResults
  VAR_INPUT
    index : UINT;
    noOfBytes : UDINT;
    value1Byte : USINT;
    value2Bytes : UINT;
    value4Bytes : UDINT;
  END_VAR
                  write := THIS^.processes.write.request(
    index := index,
    noOfBytes := noOfBytes,
    value1Byte := value1Byte,
    value2Bytes := value2Bytes,
    value4Bytes := value4Bytes);

                
END_METHOD

{attribute 'TcRpcEnable' := '1'}
METHOD update : RequestResults
                  update := THIS^.processes.update.request();

                
END_METHOD

{attribute 'TcRpcEnable' := '1'}
METHOD reset : RequestResults
                  reset := THIS^.processes.reset.request();

                
END_METHOD

{attribute 'TcRpcEnable' := '1'}
METHOD acknowledgeSafetyError : RequestResults
                  acknowledgeSafetyError := THIS^.processes.acknowledgeSafetyError.request();

                
END_METHOD

{attribute 'TcRpcEnable' := '1'}
METHOD setBrake : RequestResults
  VAR_INPUT
    newState : DriveBrakeStates;
  END_VAR
                  setBrake := THIS^.processes.setBrake.request( newState := newState );

                
END_METHOD

{attribute 'TcRpcEnable' := '1'}
METHOD _log : BOOL
  VAR_INPUT
    name : STRING;  (* Name of this function block instance *)
  END_VAR
  VAR_IN_OUT
    buffer : LogBuffer;  (* Buffer to write all logging to *)
  END_VAR
  VAR
    subBuffer : LogBuffer;  (* Temporary buffer to write logging by parts (sub-statemachines) to *)
  END_VAR
                  LOGGER(
    name := name,
    actualStatus := THIS^.actualStatus,
    previousStatus := THIS^.previousStatus,
    buffer := buffer,
    subBuffer := subBuffer,
    pHealthStatus := ADR(THIS^.statuses.healthStatus),
    pBusyStatus := ADR(THIS^.statuses.busyStatus));

                
END_METHOD
END_FUNCTION_BLOCK

FUNCTION_BLOCK SM_AX52XXDrive
  VAR_INPUT
    {attribute 'OPC.UA.DA' := '0'}
    isEnabled : BOOL;  (* Is control enabled? *)
  END_VAR
  VAR_OUTPUT
    {attribute 'OPC.UA.DA' := '1'}
    {attribute 'OPC.UA.DA.Access' := '1'}
    actualStatus : STRING;  (* Current status description *)
    previousStatus : STRING;  (* Previous status description *)
    statuses : AX52XXDriveStatuses;  (* Statuses of the state machine *)
    parts : AX52XXDriveParts;  (* Parts of the state machine *)
  END_VAR

            parts.channelA( isEnabled := isEnabled );
parts.channelB( isEnabled := isEnabled );
statuses.busyStatus( isBusy := parts.channelA.statuses.healthStatus.hasWarning OR parts.channelB.statuses.healthStatus.hasWarning );
statuses.healthStatus(
    isGood := parts.channelA.statuses.healthStatus.isGood AND parts.channelB.statuses.healthStatus.isGood,
    hasWarning := parts.channelA.statuses.healthStatus.hasWarning OR parts.channelB.statuses.healthStatus.hasWarning);

          

{attribute 'TcRpcEnable' := '1'}
METHOD _log : BOOL
  VAR_INPUT
    name : STRING;  (* Name of this function block instance *)
  END_VAR
  VAR_IN_OUT
    buffer : LogBuffer;  (* Buffer to write all logging to *)
  END_VAR
  VAR
    subBuffer : LogBuffer;  (* Temporary buffer to write logging by parts (sub-statemachines) to *)
  END_VAR
                  THIS^.parts.channelA._log(
    name := 'channelA',
    buffer := subBuffer);
THIS^.parts.channelB._log(
    name := 'channelB',
    buffer := subBuffer);
LOGGER(
    name := name,
    actualStatus := THIS^.actualStatus,
    previousStatus := THIS^.previousStatus,
    buffer := buffer,
    subBuffer := subBuffer,
    pHealthStatus := ADR(THIS^.statuses.healthStatus),
    pBusyStatus := ADR(THIS^.statuses.busyStatus));

                
END_METHOD
END_FUNCTION_BLOCK

FUNCTION_BLOCK SM_SSIEncoder
  VAR_INPUT
    {attribute 'OPC.UA.DA' := '0'}
    counterValue AT %I* : UDINT;  (* Counter value *)
    {attribute 'OPC.UA.DA' := '0'}
    status AT %I* : UINT;  (* Status *)
  END_VAR
  VAR_OUTPUT
    {attribute 'OPC.UA.DA' := '1'}
    {attribute 'OPC.UA.DA.Access' := '1'}
    actualStatus : STRING;  (* Current status description *)
    previousStatus : STRING;  (* Previous status description *)
    {attribute 'OPC.UA.DA' := '1'}
    {attribute 'OPC.UA.DA.Access' := '1'}
    dataError AT %I* : BOOL;  (* Data error *)
    {attribute 'OPC.UA.DA' := '1'}
    {attribute 'OPC.UA.DA.Access' := '1'}
    frameError AT %I* : BOOL;  (* Frame error *)
    {attribute 'OPC.UA.DA' := '1'}
    {attribute 'OPC.UA.DA.Access' := '1'}
    powerFailure AT %I* : BOOL;  (* Power failure *)
    {attribute 'OPC.UA.DA' := '1'}
    {attribute 'OPC.UA.DA.Access' := '1'}
    syncError AT %I* : BOOL;  (* Sync error *)
    statuses : SSIEncoderStatuses;  (* Statuses of the state machine *)
  END_VAR

            statuses.healthStatus( isGood := NOT(dataError OR (frameError OR (powerFailure OR syncError))) );

          

{attribute 'TcRpcEnable' := '1'}
METHOD _log : BOOL
  VAR_INPUT
    name : STRING;  (* Name of this function block instance *)
  END_VAR
  VAR_IN_OUT
    buffer : LogBuffer;  (* Buffer to write all logging to *)
  END_VAR
  VAR
    subBuffer : LogBuffer;  (* Temporary buffer to write logging by parts (sub-statemachines) to *)
  END_VAR
                  LOGGER(
    name := name,
    actualStatus := THIS^.actualStatus,
    previousStatus := THIS^.previousStatus,
    buffer := buffer,
    subBuffer := subBuffer,
    pHealthStatus := ADR(THIS^.statuses.healthStatus));

                
END_METHOD
END_FUNCTION_BLOCK

FUNCTION_BLOCK SM_IncrementalEncoder
  VAR_INPUT
    {attribute 'OPC.UA.DA' := '0'}
    isEnabled : BOOL;  (* Is control enabled? *)
    {attribute 'OPC.UA.DA' := '0'}
    counterValue AT %I* : UDINT;  (* Actual counter value *)
    {attribute 'OPC.UA.DA' := '0'}
    status AT %I* : UINT;  (* Status *)
    {attribute 'OPC.UA.DA' := '0'}
    setCounterValue AT %Q* : UDINT;  (* Counter value to be set *)
    {attribute 'OPC.UA.DA' := '0'}
    setCounter AT %Q* : BOOL;  (* Counter value to be set *)
    {attribute 'OPC.UA.DA' := '0'}
    enableLatchC AT %Q* : BOOL;  (* Enable latch C *)
  END_VAR
  VAR_OUTPUT
    {attribute 'OPC.UA.DA' := '1'}
    {attribute 'OPC.UA.DA.Access' := '1'}
    actualStatus : STRING;  (* Current status description *)
    previousStatus : STRING;  (* Previous status description *)
    {attribute 'OPC.UA.DA' := '1'}
    {attribute 'OPC.UA.DA.Access' := '1'}
    latchCValid : BOOL;  (* Bit 0: Latch C valid *)
    {attribute 'OPC.UA.DA' := '1'}
    {attribute 'OPC.UA.DA.Access' := '1'}
    latchExternValid : BOOL;  (* Bit 1: Latch extern valid *)
    {attribute 'OPC.UA.DA' := '1'}
    {attribute 'OPC.UA.DA.Access' := '1'}
    setCounterDone : BOOL;  (* Bit 2: Set counter done *)
    {attribute 'OPC.UA.DA' := '1'}
    {attribute 'OPC.UA.DA.Access' := '1'}
    counterUnderflow : BOOL;  (* Bit 3: Counter undeflow *)
    {attribute 'OPC.UA.DA' := '1'}
    {attribute 'OPC.UA.DA.Access' := '1'}
    counterOverflow : BOOL;  (* Bit 4: Counter overflow *)
    {attribute 'OPC.UA.DA' := '1'}
    {attribute 'OPC.UA.DA.Access' := '1'}
    statusOfInputStatus : BOOL;  (* Bit 5: Status of input status *)
    {attribute 'OPC.UA.DA' := '1'}
    {attribute 'OPC.UA.DA.Access' := '1'}
    openCircuit : BOOL;  (* Bit 6: Open circuit *)
    {attribute 'OPC.UA.DA' := '1'}
    {attribute 'OPC.UA.DA.Access' := '1'}
    extrapolationStall : BOOL;  (* Bit 7: Extrapolation stall *)
    {attribute 'OPC.UA.DA' := '1'}
    {attribute 'OPC.UA.DA.Access' := '1'}
    statusOfInputA : BOOL;  (* Bit 8: Status of input A *)
    {attribute 'OPC.UA.DA' := '1'}
    {attribute 'OPC.UA.DA.Access' := '1'}
    statusOfInputB : BOOL;  (* Bit 9: Status of input B *)
    {attribute 'OPC.UA.DA' := '1'}
    {attribute 'OPC.UA.DA.Access' := '1'}
    statusOfInputC : BOOL;  (* Bit 10: Status of input C *)
    {attribute 'OPC.UA.DA' := '1'}
    {attribute 'OPC.UA.DA.Access' := '1'}
    statusOfInputGate : BOOL;  (* Bit 11: Status of input gate *)
    {attribute 'OPC.UA.DA' := '1'}
    {attribute 'OPC.UA.DA.Access' := '1'}
    statusOfExternLatch : BOOL;  (* Bit 12: Status of external latch *)
    {attribute 'OPC.UA.DA' := '1'}
    {attribute 'OPC.UA.DA.Access' := '1'}
    syncError : BOOL;  (* Bit 13: Sync error *)
    statuses : IncrementalEncoderStatuses;  (* Statuses of the state machine *)
    processes : IncrementalEncoderProcesses;  (* Processes of the state machine *)
  END_VAR

            statuses.healthStatus( isGood := NOT((NOT(statusOfInputStatus)) OR (openCircuit OR (extrapolationStall OR syncError))) );
statuses.busyStatus( isBusy := processes.enableCounterResetC.statuses.busyStatus.busy OR processes.disableCounterResetC.statuses.busyStatus.busy );
processes.enableCounterResetC( isEnabled := isEnabled );
processes.disableCounterResetC( isEnabled := isEnabled );

          

{attribute 'TcRpcEnable' := '1'}
METHOD enableCounterResetC : RequestResults
                  enableCounterResetC := THIS^.processes.enableCounterResetC.request();

                
END_METHOD

{attribute 'TcRpcEnable' := '1'}
METHOD disableCounterResetC : RequestResults
                  disableCounterResetC := THIS^.processes.disableCounterResetC.request();

                
END_METHOD

{attribute 'TcRpcEnable' := '1'}
METHOD _log : BOOL
  VAR_INPUT
    name : STRING;  (* Name of this function block instance *)
  END_VAR
  VAR_IN_OUT
    buffer : LogBuffer;  (* Buffer to write all logging to *)
  END_VAR
  VAR
    subBuffer : LogBuffer;  (* Temporary buffer to write logging by parts (sub-statemachines) to *)
  END_VAR
                  LOGGER(
    name := name,
    actualStatus := THIS^.actualStatus,
    previousStatus := THIS^.previousStatus,
    buffer := buffer,
    subBuffer := subBuffer,
    pHealthStatus := ADR(THIS^.statuses.healthStatus),
    pBusyStatus := ADR(THIS^.statuses.busyStatus));

                
END_METHOD
END_FUNCTION_BLOCK

FUNCTION_BLOCK SM_EtherCatDevice
  VAR_INPUT
    {attribute 'OPC.UA.DA' := '1'}
    {attribute 'OPC.UA.DA.Access' := '1'}
    id : STRING;  (* Label according to the electric schemes *)
    {attribute 'OPC.UA.DA' := '1'}
    {attribute 'OPC.UA.DA.Access' := '1'}
    typeId : STRING;  (* Manufacturer type, e.g. EL1008 *)
    {attribute 'OPC.UA.DA' := '1'}
    {attribute 'OPC.UA.DA.Access' := '1'}
    wcState AT %I* : BOOL;  (* 0 = Data valid, 1 = Data invalid *)
    {attribute 'OPC.UA.DA' := '1'}
    {attribute 'OPC.UA.DA.Access' := '1'}
    infoData AT %I* : UINT;  (* EtherCAT state *)
  END_VAR
  VAR_OUTPUT
    {attribute 'OPC.UA.DA' := '1'}
    {attribute 'OPC.UA.DA.Access' := '1'}
    actualStatus : STRING;  (* Current status description *)
    previousStatus : STRING;  (* Previous status description *)
    statuses : EtherCatDeviceStatuses;  (* Statuses of the state machine *)
  END_VAR

            statuses.healthStatus( isGood := (wcState = FALSE) AND (infoData = 8) );

          

{attribute 'TcRpcEnable' := '1'}
METHOD _log : BOOL
  VAR_INPUT
    name : STRING;  (* Name of this function block instance *)
  END_VAR
  VAR_IN_OUT
    buffer : LogBuffer;  (* Buffer to write all logging to *)
  END_VAR
  VAR
    subBuffer : LogBuffer;  (* Temporary buffer to write logging by parts (sub-statemachines) to *)
  END_VAR
                  LOGGER(
    name := name,
    actualStatus := THIS^.actualStatus,
    previousStatus := THIS^.previousStatus,
    buffer := buffer,
    subBuffer := subBuffer,
    pHealthStatus := ADR(THIS^.statuses.healthStatus));

                
END_METHOD
END_FUNCTION_BLOCK

FUNCTION_BLOCK SM_CANopenBus
  VAR_INPUT
    {attribute 'OPC.UA.DA' := '1'}
    {attribute 'OPC.UA.DA.Access' := '1'}
    error AT %I* : USINT;  (* Number of boxes with BoxState unequal to 0 *)
    {attribute 'OPC.UA.DA' := '1'}
    {attribute 'OPC.UA.DA.Access' := '1'}
    canState AT %I* : UINT;  (* CAN state (See system manager for bit interpretation *)
    {attribute 'OPC.UA.DA' := '1'}
    {attribute 'OPC.UA.DA.Access' := '1'}
    rxErrorCounter AT %I* : USINT;  (* RxError-counter of the CAN controller *)
    {attribute 'OPC.UA.DA' := '1'}
    {attribute 'OPC.UA.DA.Access' := '1'}
    txErrorCounter AT %I* : USINT;  (* TxError-counter of the CAN controller *)
  END_VAR
  VAR_OUTPUT
    {attribute 'OPC.UA.DA' := '1'}
    {attribute 'OPC.UA.DA.Access' := '1'}
    actualStatus : STRING;  (* Current status description *)
    previousStatus : STRING;  (* Previous status description *)
    statuses : CANopenBusStatuses;  (* Statuses of the state machine *)
  END_VAR

            statuses.healthStatus( isGood := error = 0 );

          

{attribute 'TcRpcEnable' := '1'}
METHOD _log : BOOL
  VAR_INPUT
    name : STRING;  (* Name of this function block instance *)
  END_VAR
  VAR_IN_OUT
    buffer : LogBuffer;  (* Buffer to write all logging to *)
  END_VAR
  VAR
    subBuffer : LogBuffer;  (* Temporary buffer to write logging by parts (sub-statemachines) to *)
  END_VAR
                  LOGGER(
    name := name,
    actualStatus := THIS^.actualStatus,
    previousStatus := THIS^.previousStatus,
    buffer := buffer,
    subBuffer := subBuffer,
    pHealthStatus := ADR(THIS^.statuses.healthStatus));

                
END_METHOD
END_FUNCTION_BLOCK

FUNCTION_BLOCK SM_CurrentMeasurement
  VAR_INPUT
    {attribute 'OPC.UA.DA' := '0'}
    microAmpsValue AT %I* : DINT;  (* Measured current in microamps *)
    {attribute 'OPC.UA.DA' := '0'}
    error AT %I* : BOOL;  (* Error *)
  END_VAR
  VAR_OUTPUT
    {attribute 'OPC.UA.DA' := '1'}
    {attribute 'OPC.UA.DA.Access' := '1'}
    actualStatus : STRING;  (* Current status description *)
    previousStatus : STRING;  (* Previous status description *)
    {attribute 'OPC.UA.DA' := '1'}
    {attribute 'OPC.UA.DA.Access' := '1'}
    current : Current;  (* The measured current *)
    statuses : CurrentMeasurementStatuses;  (* Statuses of the state machine *)
  END_VAR

            current( newAmpsValue := microAmpsValue / 1000000.0 );
statuses.healthStatus( isGood := NOT(error) );

          

{attribute 'TcRpcEnable' := '1'}
METHOD _log : BOOL
  VAR_INPUT
    name : STRING;  (* Name of this function block instance *)
  END_VAR
  VAR_IN_OUT
    buffer : LogBuffer;  (* Buffer to write all logging to *)
  END_VAR
  VAR
    subBuffer : LogBuffer;  (* Temporary buffer to write logging by parts (sub-statemachines) to *)
  END_VAR
                  LOGGER(
    name := name,
    actualStatus := THIS^.actualStatus,
    previousStatus := THIS^.previousStatus,
    buffer := buffer,
    subBuffer := subBuffer,
    pHealthStatus := ADR(THIS^.statuses.healthStatus));

                
END_METHOD
END_FUNCTION_BLOCK

FUNCTION_BLOCK SM_VoltageMeasurement
  VAR_INPUT
    {attribute 'OPC.UA.DA' := '0'}
    rawValue AT %I* : INT;  (* Measured raw value *)
    {attribute 'OPC.UA.DA' := '0'}
    error AT %I* : BOOL;  (* Error *)
    {attribute 'OPC.UA.DA' := '0'}
    conversionFactor : LREAL := 0.00030517578125;  (* rawValue * conversionFactor = volt.value *)
  END_VAR
  VAR_OUTPUT
    {attribute 'OPC.UA.DA' := '1'}
    {attribute 'OPC.UA.DA.Access' := '1'}
    actualStatus : STRING;  (* Current status description *)
    previousStatus : STRING;  (* Previous status description *)
    {attribute 'OPC.UA.DA' := '1'}
    {attribute 'OPC.UA.DA.Access' := '1'}
    actual : Voltage;  (* Actual value *)
    {attribute 'OPC.UA.DA' := '1'}
    {attribute 'OPC.UA.DA.Access' := '1'}
    average : Voltage;  (* Moving average value *)
    {attribute 'OPC.UA.DA' := '1'}
    {attribute 'OPC.UA.DA.Access' := '1'}
    underrange AT %I* : BOOL;  (* Underrange *)
    {attribute 'OPC.UA.DA' := '1'}
    {attribute 'OPC.UA.DA.Access' := '1'}
    overrange AT %I* : BOOL;  (* Overrange *)
    statuses : VoltageMeasurementStatuses;  (* Statuses of the state machine *)
  END_VAR
  VAR_IN_OUT
    {attribute 'OPC.UA.DA' := '0'}
    config : MeasurementConfig;  (* Reference to the config (alarms in volts) *)
  END_VAR

            actual( newVoltValue := (rawValue * conversionFactor) + config.offset );
statuses.enabledStatus( isEnabled := config.enabled );
statuses.healthStatus(
    superState := statuses.enabledStatus.enabled,
    isGood := NOT(error OR (underrange OR (overrange OR (statuses.alarmStatus.hiHi OR statuses.alarmStatus.loLo)))),
    hasWarning := statuses.alarmStatus.hi OR statuses.alarmStatus.lo);
statuses.alarmStatus(
    superState := statuses.enabledStatus.enabled,
    config := config.alarms,
    value := average.volt.value);

          

{attribute 'TcRpcEnable' := '1'}
METHOD _log : BOOL
  VAR_INPUT
    name : STRING;  (* Name of this function block instance *)
  END_VAR
  VAR_IN_OUT
    buffer : LogBuffer;  (* Buffer to write all logging to *)
  END_VAR
  VAR
    subBuffer : LogBuffer;  (* Temporary buffer to write logging by parts (sub-statemachines) to *)
  END_VAR
                  LOGGER(
    name := name,
    actualStatus := THIS^.actualStatus,
    previousStatus := THIS^.previousStatus,
    buffer := buffer,
    subBuffer := subBuffer,
    pHealthStatus := ADR(THIS^.statuses.healthStatus));

                
END_METHOD
END_FUNCTION_BLOCK

FUNCTION_BLOCK SM_TemperatureMeasurement
  VAR_INPUT
    {attribute 'OPC.UA.DA' := '0'}
    rawValue AT %I* : INT;  (* Measured raw value *)
    {attribute 'OPC.UA.DA' := '0'}
    error AT %I* : BOOL;  (* Error *)
    {attribute 'OPC.UA.DA' := '0'}
    conversionFactor : LREAL := 0.01;  (* rawValue * conversionFactor = temperature.degrees.value *)
  END_VAR
  VAR_OUTPUT
    {attribute 'OPC.UA.DA' := '1'}
    {attribute 'OPC.UA.DA.Access' := '1'}
    actualStatus : STRING;  (* Current status description *)
    previousStatus : STRING;  (* Previous status description *)
    {attribute 'OPC.UA.DA' := '1'}
    {attribute 'OPC.UA.DA.Access' := '1'}
    actual : Temperature;  (* Actual value *)
    {attribute 'OPC.UA.DA' := '1'}
    {attribute 'OPC.UA.DA.Access' := '1'}
    average : Temperature;  (* Moving average value *)
    {attribute 'OPC.UA.DA' := '1'}
    {attribute 'OPC.UA.DA.Access' := '1'}
    underrange AT %I* : BOOL;  (* Underrange *)
    {attribute 'OPC.UA.DA' := '1'}
    {attribute 'OPC.UA.DA.Access' := '1'}
    overrange AT %I* : BOOL;  (* Overrange *)
    statuses : TemperatureMeasurementStatuses;  (* Statuses of the state machine *)
  END_VAR
  VAR_IN_OUT
    {attribute 'OPC.UA.DA' := '0'}
    config : MeasurementConfig;  (* Reference to the config (alarms in degrees celsius) *)
  END_VAR

            actual( newCelsiusValue := (rawValue * conversionFactor) + config.offset );
statuses.enabledStatus( isEnabled := config.enabled );
statuses.healthStatus(
    superState := statuses.enabledStatus.enabled,
    isGood := NOT(error OR (underrange OR (overrange OR (statuses.alarmStatus.hiHi OR statuses.alarmStatus.loLo)))),
    hasWarning := statuses.alarmStatus.hi OR statuses.alarmStatus.lo);
statuses.alarmStatus(
    superState := statuses.enabledStatus.enabled,
    config := config.alarms,
    value := average.celsius.value);

          

{attribute 'TcRpcEnable' := '1'}
METHOD _log : BOOL
  VAR_INPUT
    name : STRING;  (* Name of this function block instance *)
  END_VAR
  VAR_IN_OUT
    buffer : LogBuffer;  (* Buffer to write all logging to *)
  END_VAR
  VAR
    subBuffer : LogBuffer;  (* Temporary buffer to write logging by parts (sub-statemachines) to *)
  END_VAR
                  LOGGER(
    name := name,
    actualStatus := THIS^.actualStatus,
    previousStatus := THIS^.previousStatus,
    buffer := buffer,
    subBuffer := subBuffer,
    pHealthStatus := ADR(THIS^.statuses.healthStatus));

                
END_METHOD
END_FUNCTION_BLOCK

FUNCTION_BLOCK SM_PressureMeasurement
  VAR_INPUT
    {attribute 'OPC.UA.DA' := '0'}
    rawValue AT %I* : INT;  (* Measured raw value *)
    {attribute 'OPC.UA.DA' := '0'}
    error AT %I* : BOOL;  (* Error *)
    {attribute 'OPC.UA.DA' := '0'}
    conversionFactor : LREAL := 1.0;  (* rawValue * conversionFactor = bar.value *)
  END_VAR
  VAR_OUTPUT
    {attribute 'OPC.UA.DA' := '1'}
    {attribute 'OPC.UA.DA.Access' := '1'}
    actualStatus : STRING;  (* Current status description *)
    previousStatus : STRING;  (* Previous status description *)
    {attribute 'OPC.UA.DA' := '1'}
    {attribute 'OPC.UA.DA.Access' := '1'}
    actual : Pressure;  (* Actual value *)
    {attribute 'OPC.UA.DA' := '1'}
    {attribute 'OPC.UA.DA.Access' := '1'}
    average : Pressure;  (* Moving average value *)
    {attribute 'OPC.UA.DA' := '1'}
    {attribute 'OPC.UA.DA.Access' := '1'}
    underrange AT %I* : BOOL;  (* Underrange *)
    {attribute 'OPC.UA.DA' := '1'}
    {attribute 'OPC.UA.DA.Access' := '1'}
    overrange AT %I* : BOOL;  (* Overrange *)
    statuses : PressureMeasurementStatuses;  (* Statuses of the state machine *)
  END_VAR
  VAR_IN_OUT
    {attribute 'OPC.UA.DA' := '0'}
    config : MeasurementConfig;  (* Reference to the config (alarms in bar) *)
  END_VAR

            actual( newBarValue := (rawValue * conversionFactor) + config.offset );
statuses.enabledStatus( isEnabled := config.enabled );
statuses.healthStatus(
    superState := statuses.enabledStatus.enabled,
    isGood := NOT(error OR (underrange OR (overrange OR (statuses.alarmStatus.hiHi OR statuses.alarmStatus.loLo)))),
    hasWarning := statuses.alarmStatus.hi OR statuses.alarmStatus.lo);
statuses.alarmStatus(
    superState := statuses.enabledStatus.enabled,
    config := config.alarms,
    value := average.bar.value);

          

{attribute 'TcRpcEnable' := '1'}
METHOD _log : BOOL
  VAR_INPUT
    name : STRING;  (* Name of this function block instance *)
  END_VAR
  VAR_IN_OUT
    buffer : LogBuffer;  (* Buffer to write all logging to *)
  END_VAR
  VAR
    subBuffer : LogBuffer;  (* Temporary buffer to write logging by parts (sub-statemachines) to *)
  END_VAR
                  LOGGER(
    name := name,
    actualStatus := THIS^.actualStatus,
    previousStatus := THIS^.previousStatus,
    buffer := buffer,
    subBuffer := subBuffer,
    pHealthStatus := ADR(THIS^.statuses.healthStatus));

                
END_METHOD
END_FUNCTION_BLOCK

FUNCTION_BLOCK SM_FrequencyMeasurement
  VAR_INPUT
    {attribute 'OPC.UA.DA' := '0'}
    rawValue AT %I* : INT;  (* Measured raw value *)
    {attribute 'OPC.UA.DA' := '0'}
    error AT %I* : BOOL;  (* Error *)
    {attribute 'OPC.UA.DA' := '0'}
    conversionFactor : LREAL := 1.0;  (* rawValue * conversionFactor = hertz.value *)
  END_VAR
  VAR_OUTPUT
    {attribute 'OPC.UA.DA' := '1'}
    {attribute 'OPC.UA.DA.Access' := '1'}
    actualStatus : STRING;  (* Current status description *)
    previousStatus : STRING;  (* Previous status description *)
    {attribute 'OPC.UA.DA' := '1'}
    {attribute 'OPC.UA.DA.Access' := '1'}
    actual : Frequency;  (* Actual value *)
    {attribute 'OPC.UA.DA' := '1'}
    {attribute 'OPC.UA.DA.Access' := '1'}
    average : Frequency;  (* Moving average value *)
    {attribute 'OPC.UA.DA' := '1'}
    {attribute 'OPC.UA.DA.Access' := '1'}
    underrange AT %I* : BOOL;  (* Underrange *)
    {attribute 'OPC.UA.DA' := '1'}
    {attribute 'OPC.UA.DA.Access' := '1'}
    overrange AT %I* : BOOL;  (* Overrange *)
    statuses : FrequencyMeasurementStatuses;  (* Statuses of the state machine *)
  END_VAR
  VAR_IN_OUT
    {attribute 'OPC.UA.DA' := '0'}
    config : MeasurementConfig;  (* Reference to the config (alarms in hertz) *)
  END_VAR

            actual( newHertzValue := (rawValue * conversionFactor) + config.offset );
statuses.enabledStatus( isEnabled := config.enabled );
statuses.healthStatus(
    superState := statuses.enabledStatus.enabled,
    isGood := NOT(error OR (underrange OR (overrange OR (statuses.alarmStatus.hiHi OR statuses.alarmStatus.loLo)))),
    hasWarning := statuses.alarmStatus.hi OR statuses.alarmStatus.lo);
statuses.alarmStatus(
    superState := statuses.enabledStatus.enabled,
    config := config.alarms,
    value := average.hertz.value);

          

{attribute 'TcRpcEnable' := '1'}
METHOD _log : BOOL
  VAR_INPUT
    name : STRING;  (* Name of this function block instance *)
  END_VAR
  VAR_IN_OUT
    buffer : LogBuffer;  (* Buffer to write all logging to *)
  END_VAR
  VAR
    subBuffer : LogBuffer;  (* Temporary buffer to write logging by parts (sub-statemachines) to *)
  END_VAR
                  LOGGER(
    name := name,
    actualStatus := THIS^.actualStatus,
    previousStatus := THIS^.previousStatus,
    buffer := buffer,
    subBuffer := subBuffer,
    pHealthStatus := ADR(THIS^.statuses.healthStatus));

                
END_METHOD
END_FUNCTION_BLOCK

FUNCTION_BLOCK SM_GForceMeasurement
  VAR_INPUT
    {attribute 'OPC.UA.DA' := '0'}
    milliGValue AT %I* : INT;  (* Measured raw milliG value (linked to I/O module) *)
    {attribute 'OPC.UA.DA' := '0'}
    error AT %I* : BOOL;  (* Error *)
  END_VAR
  VAR_OUTPUT
    {attribute 'OPC.UA.DA' := '1'}
    {attribute 'OPC.UA.DA.Access' := '1'}
    actualStatus : STRING;  (* Current status description *)
    previousStatus : STRING;  (* Previous status description *)
    {attribute 'OPC.UA.DA' := '1'}
    {attribute 'OPC.UA.DA.Access' := '1'}
    actual : GForce;  (* Actual value *)
    {attribute 'OPC.UA.DA' := '1'}
    {attribute 'OPC.UA.DA.Access' := '1'}
    average : GForce;  (* Moving average value *)
    statuses : GForceMeasurementStatuses;  (* Statuses of the state machine *)
  END_VAR

            actual( newMilliGValue := milliGValue );
statuses.healthStatus( isGood := NOT(error) );

          

{attribute 'TcRpcEnable' := '1'}
METHOD _log : BOOL
  VAR_INPUT
    name : STRING;  (* Name of this function block instance *)
  END_VAR
  VAR_IN_OUT
    buffer : LogBuffer;  (* Buffer to write all logging to *)
  END_VAR
  VAR
    subBuffer : LogBuffer;  (* Temporary buffer to write logging by parts (sub-statemachines) to *)
  END_VAR
                  LOGGER(
    name := name,
    actualStatus := THIS^.actualStatus,
    previousStatus := THIS^.previousStatus,
    buffer := buffer,
    subBuffer := subBuffer,
    pHealthStatus := ADR(THIS^.statuses.healthStatus));

                
END_METHOD
END_FUNCTION_BLOCK

FUNCTION_BLOCK SM_RelativeHumidityMeasurement
  VAR_INPUT
    {attribute 'OPC.UA.DA' := '0'}
    rawValue AT %I* : INT;  (* Measured raw value *)
    {attribute 'OPC.UA.DA' := '0'}
    error AT %I* : BOOL;  (* Error *)
    {attribute 'OPC.UA.DA' := '0'}
    conversionFactor : LREAL := 3.0518509476E-05;  (* rawValue * conversionFactor = fraction.value *)
  END_VAR
  VAR_OUTPUT
    {attribute 'OPC.UA.DA' := '1'}
    {attribute 'OPC.UA.DA.Access' := '1'}
    actualStatus : STRING;  (* Current status description *)
    previousStatus : STRING;  (* Previous status description *)
    {attribute 'OPC.UA.DA' := '1'}
    {attribute 'OPC.UA.DA.Access' := '1'}
    actual : Fraction;  (* Actual value *)
    {attribute 'OPC.UA.DA' := '1'}
    {attribute 'OPC.UA.DA.Access' := '1'}
    average : Fraction;  (* Moving average value *)
    {attribute 'OPC.UA.DA' := '1'}
    {attribute 'OPC.UA.DA.Access' := '1'}
    underrange AT %I* : BOOL;  (* Underrange *)
    {attribute 'OPC.UA.DA' := '1'}
    {attribute 'OPC.UA.DA.Access' := '1'}
    overrange AT %I* : BOOL;  (* Overrange *)
    statuses : RelativeHumidityMeasurementStatuses;  (* Statuses of the state machine *)
  END_VAR
  VAR_IN_OUT
    {attribute 'OPC.UA.DA' := '0'}
    config : MeasurementConfig;  (* Reference to the config (alarms in percent) *)
  END_VAR

            actual( newFractionValue := (rawValue * conversionFactor) + config.offset );
statuses.enabledStatus( isEnabled := config.enabled );
statuses.healthStatus(
    superState := statuses.enabledStatus.enabled,
    isGood := NOT(error OR (underrange OR (overrange OR (statuses.alarmStatus.hiHi OR statuses.alarmStatus.loLo)))),
    hasWarning := statuses.alarmStatus.hi OR statuses.alarmStatus.lo);
statuses.alarmStatus(
    superState := statuses.enabledStatus.enabled,
    config := config.alarms,
    value := average.percent.value);

          

{attribute 'TcRpcEnable' := '1'}
METHOD _log : BOOL
  VAR_INPUT
    name : STRING;  (* Name of this function block instance *)
  END_VAR
  VAR_IN_OUT
    buffer : LogBuffer;  (* Buffer to write all logging to *)
  END_VAR
  VAR
    subBuffer : LogBuffer;  (* Temporary buffer to write logging by parts (sub-statemachines) to *)
  END_VAR
                  LOGGER(
    name := name,
    actualStatus := THIS^.actualStatus,
    previousStatus := THIS^.previousStatus,
    buffer := buffer,
    subBuffer := subBuffer,
    pHealthStatus := ADR(THIS^.statuses.healthStatus));

                
END_METHOD
END_FUNCTION_BLOCK

FUNCTION_BLOCK SM_ForceMeasurement
  VAR_INPUT
    {attribute 'OPC.UA.DA' := '0'}
    rawValue AT %I* : DINT;  (* Measured raw value *)
    {attribute 'OPC.UA.DA' := '0'}
    error AT %I* : BOOL;  (* Error *)
    {attribute 'OPC.UA.DA' := '0'}
    underrange AT %I* : BOOL;  (* Underrange *)
    {attribute 'OPC.UA.DA' := '0'}
    overrange AT %I* : BOOL;  (* Overrange *)
    {attribute 'OPC.UA.DA' := '0'}
    conversionFactor : LREAL := 1.0;  (* rawValue * conversionFactor = newton.value *)
  END_VAR
  VAR_OUTPUT
    {attribute 'OPC.UA.DA' := '1'}
    {attribute 'OPC.UA.DA.Access' := '1'}
    actualStatus : STRING;  (* Current status description *)
    previousStatus : STRING;  (* Previous status description *)
    {attribute 'OPC.UA.DA' := '1'}
    {attribute 'OPC.UA.DA.Access' := '1'}
    actual : Force;  (* Actual value *)
    {attribute 'OPC.UA.DA' := '1'}
    {attribute 'OPC.UA.DA.Access' := '1'}
    average : Force;  (* Moving average value *)
    statuses : ForceMeasurementStatuses;  (* Statuses of the state machine *)
  END_VAR
  VAR_IN_OUT
    {attribute 'OPC.UA.DA' := '0'}
    config : MeasurementConfig;  (* Reference to the config (alarms in Newton) *)
  END_VAR

            actual( newNewtonValue := (rawValue * conversionFactor) + config.offset );
statuses.enabledStatus( isEnabled := config.enabled );
statuses.healthStatus(
    superState := statuses.enabledStatus.enabled,
    isGood := NOT(error OR (underrange OR (overrange OR (statuses.alarmStatus.hiHi OR statuses.alarmStatus.loLo)))),
    hasWarning := statuses.alarmStatus.hi OR statuses.alarmStatus.lo);
statuses.alarmStatus(
    superState := statuses.enabledStatus.enabled,
    config := config.alarms,
    value := average.newton.value);

          

{attribute 'TcRpcEnable' := '1'}
METHOD _log : BOOL
  VAR_INPUT
    name : STRING;  (* Name of this function block instance *)
  END_VAR
  VAR_IN_OUT
    buffer : LogBuffer;  (* Buffer to write all logging to *)
  END_VAR
  VAR
    subBuffer : LogBuffer;  (* Temporary buffer to write logging by parts (sub-statemachines) to *)
  END_VAR
                  LOGGER(
    name := name,
    actualStatus := THIS^.actualStatus,
    previousStatus := THIS^.previousStatus,
    buffer := buffer,
    subBuffer := subBuffer,
    pHealthStatus := ADR(THIS^.statuses.healthStatus));

                
END_METHOD
END_FUNCTION_BLOCK

FUNCTION_BLOCK SM_LinearPositionMeasurement16
  VAR_INPUT
    {attribute 'OPC.UA.DA' := '0'}
    rawValue AT %I* : INT;  (* Measured raw value *)
    {attribute 'OPC.UA.DA' := '0'}
    error AT %I* : BOOL;  (* Error *)
    {attribute 'OPC.UA.DA' := '0'}
    underrange AT %I* : BOOL;  (* Underrange *)
    {attribute 'OPC.UA.DA' := '0'}
    overrange AT %I* : BOOL;  (* Overrange *)
    {attribute 'OPC.UA.DA' := '0'}
    conversionFactor : LREAL := 3.0518509476E-05;  (* rawValue * conversionFactor = millimeters.value *)
  END_VAR
  VAR_OUTPUT
    {attribute 'OPC.UA.DA' := '1'}
    {attribute 'OPC.UA.DA.Access' := '1'}
    actualStatus : STRING;  (* Current status description *)
    previousStatus : STRING;  (* Previous status description *)
    {attribute 'OPC.UA.DA' := '1'}
    {attribute 'OPC.UA.DA.Access' := '1'}
    actual : LinearPosition;  (* Actual value *)
    {attribute 'OPC.UA.DA' := '1'}
    {attribute 'OPC.UA.DA.Access' := '1'}
    average : LinearPosition;  (* Moving average value *)
    statuses : LinearPositionMeasurement16Statuses;  (* Statuses of the state machine *)
  END_VAR
  VAR_IN_OUT
    {attribute 'OPC.UA.DA' := '0'}
    config : MeasurementConfig;  (* Reference to the config (alarms in millimeters) *)
  END_VAR

            actual( newMillimetersValue := (rawValue * conversionFactor) + config.offset );
statuses.enabledStatus( isEnabled := config.enabled );
statuses.healthStatus(
    superState := statuses.enabledStatus.enabled,
    isGood := NOT(error OR (underrange OR (overrange OR (statuses.alarmStatus.hiHi OR statuses.alarmStatus.loLo)))),
    hasWarning := statuses.alarmStatus.hi OR statuses.alarmStatus.lo);
statuses.alarmStatus(
    superState := statuses.enabledStatus.enabled,
    config := config.alarms,
    value := average.millimeters.value);

          

{attribute 'TcRpcEnable' := '1'}
METHOD _log : BOOL
  VAR_INPUT
    name : STRING;  (* Name of this function block instance *)
  END_VAR
  VAR_IN_OUT
    buffer : LogBuffer;  (* Buffer to write all logging to *)
  END_VAR
  VAR
    subBuffer : LogBuffer;  (* Temporary buffer to write logging by parts (sub-statemachines) to *)
  END_VAR
                  LOGGER(
    name := name,
    actualStatus := THIS^.actualStatus,
    previousStatus := THIS^.previousStatus,
    buffer := buffer,
    subBuffer := subBuffer,
    pHealthStatus := ADR(THIS^.statuses.healthStatus));

                
END_METHOD
END_FUNCTION_BLOCK

FUNCTION_BLOCK SM_LinearPositionMeasurementU32
  VAR_INPUT
    {attribute 'OPC.UA.DA' := '0'}
    rawValue AT %I* : UDINT;  (* Measured raw value *)
    {attribute 'OPC.UA.DA' := '0'}
    error AT %I* : BOOL;  (* Error *)
    {attribute 'OPC.UA.DA' := '0'}
    underrange AT %I* : BOOL;  (* Underrange *)
    {attribute 'OPC.UA.DA' := '0'}
    overrange AT %I* : BOOL;  (* Overrange *)
    {attribute 'OPC.UA.DA' := '0'}
    conversionFactor : LREAL := 4.65661287525E-10;  (* rawValue * conversionFactor = millimeters.value *)
  END_VAR
  VAR_OUTPUT
    {attribute 'OPC.UA.DA' := '1'}
    {attribute 'OPC.UA.DA.Access' := '1'}
    actualStatus : STRING;  (* Current status description *)
    previousStatus : STRING;  (* Previous status description *)
    {attribute 'OPC.UA.DA' := '1'}
    {attribute 'OPC.UA.DA.Access' := '1'}
    actual : LinearPosition;  (* Actual value *)
    {attribute 'OPC.UA.DA' := '1'}
    {attribute 'OPC.UA.DA.Access' := '1'}
    average : LinearPosition;  (* Moving average value *)
    statuses : LinearPositionMeasurementU32Statuses;  (* Statuses of the state machine *)
  END_VAR
  VAR_IN_OUT
    {attribute 'OPC.UA.DA' := '0'}
    config : MeasurementConfig;  (* Reference to the config (alarms in millimeters) *)
  END_VAR

            actual( newMillimetersValue := (rawValue * conversionFactor) + config.offset );
statuses.enabledStatus( isEnabled := config.enabled );
statuses.healthStatus(
    superState := statuses.enabledStatus.enabled,
    isGood := NOT(error OR (underrange OR (overrange OR (statuses.alarmStatus.hiHi OR statuses.alarmStatus.loLo)))),
    hasWarning := statuses.alarmStatus.hi OR statuses.alarmStatus.lo);
statuses.alarmStatus(
    superState := statuses.enabledStatus.enabled,
    config := config.alarms,
    value := average.millimeters.value);

          

{attribute 'TcRpcEnable' := '1'}
METHOD _log : BOOL
  VAR_INPUT
    name : STRING;  (* Name of this function block instance *)
  END_VAR
  VAR_IN_OUT
    buffer : LogBuffer;  (* Buffer to write all logging to *)
  END_VAR
  VAR
    subBuffer : LogBuffer;  (* Temporary buffer to write logging by parts (sub-statemachines) to *)
  END_VAR
                  LOGGER(
    name := name,
    actualStatus := THIS^.actualStatus,
    previousStatus := THIS^.previousStatus,
    buffer := buffer,
    subBuffer := subBuffer,
    pHealthStatus := ADR(THIS^.statuses.healthStatus));

                
END_METHOD
END_FUNCTION_BLOCK

FUNCTION_BLOCK SM_SimpleRelay
  VAR_INPUT
    {attribute 'OPC.UA.DA' := '0'}
    isEnabled : BOOL;  (* Is control enabled? *)
  END_VAR
  VAR_OUTPUT
    {attribute 'OPC.UA.DA' := '1'}
    {attribute 'OPC.UA.DA.Access' := '1'}
    actualStatus : STRING;  (* Current status description *)
    previousStatus : STRING;  (* Previous status description *)
    {attribute 'OPC.UA.DA' := '1'}
    {attribute 'OPC.UA.DA.Access' := '1'}
    digitalOutput AT %Q* : BOOL;  (* Boolean, to bind to digital output *)
    statuses : SimpleRelayStatuses;  (* Statuses of the state machine *)
    processes : SimpleRelayProcesses;  (* Processes of the state machine *)
  END_VAR

            statuses.busyStatus( isBusy := processes.setEnabled.statuses.busyStatus.busy );
processes.setEnabled( isEnabled := isEnabled AND processes.setEnabled.statuses.busyStatus.idle );

          

{attribute 'TcRpcEnable' := '1'}
METHOD setEnabled : RequestResults
  VAR_INPUT
    enabled : BOOL;
  END_VAR
                  setEnabled := THIS^.processes.setEnabled.request( enabled := enabled );

                
END_METHOD

{attribute 'TcRpcEnable' := '1'}
METHOD _log : BOOL
  VAR_INPUT
    name : STRING;  (* Name of this function block instance *)
  END_VAR
  VAR_IN_OUT
    buffer : LogBuffer;  (* Buffer to write all logging to *)
  END_VAR
  VAR
    subBuffer : LogBuffer;  (* Temporary buffer to write logging by parts (sub-statemachines) to *)
  END_VAR
                  LOGGER(
    name := name,
    actualStatus := THIS^.actualStatus,
    previousStatus := THIS^.previousStatus,
    buffer := buffer,
    subBuffer := subBuffer,
    pBusyStatus := ADR(THIS^.statuses.busyStatus));

                
END_METHOD
END_FUNCTION_BLOCK

FUNCTION_BLOCK SM_ConfigManager
  VAR_INPUT
    {attribute 'OPC.UA.DA' := '1'}
    {attribute 'OPC.UA.DA.Access' := '1'}
    filePath : STRING;  (* Full path of the config filename *)
    {attribute 'OPC.UA.DA' := '0'}
    isEnabled : BOOL;  (* Is control enabled? *)
  END_VAR
  VAR_OUTPUT
    {attribute 'OPC.UA.DA' := '1'}
    {attribute 'OPC.UA.DA.Access' := '1'}
    actualStatus : STRING;  (* Current status description *)
    previousStatus : STRING;  (* Previous status description *)
    statuses : ConfigManagerStatuses;  (* Statuses of the state machine *)
    processes : ConfigManagerProcesses;  (* Processes of the state machine *)
  END_VAR

            statuses.busyStatus( isBusy := processes.save.statuses.busyStatus.busy OR (processes.load.statuses.busyStatus.busy OR processes.activate.statuses.busyStatus.busy) );
statuses.healthStatus(
    isGood := processes.save.statuses.healthStatus.isGood AND (processes.load.statuses.healthStatus.isGood AND processes.activate.statuses.healthStatus.isGood),
    hasWarning := processes.save.statuses.healthStatus.hasWarning OR (processes.load.statuses.healthStatus.hasWarning OR processes.activate.statuses.healthStatus.hasWarning));
processes.save( isEnabled := isEnabled AND statuses.busyStatus.idle );
processes.load( isEnabled := isEnabled AND statuses.busyStatus.idle );
processes.activate( isEnabled := isEnabled AND statuses.busyStatus.idle );

          

{attribute 'TcRpcEnable' := '1'}
METHOD save : RequestResults
  VAR_INPUT
    filePath : STRING;
  END_VAR
                  save := THIS^.processes.save.request( filePath := filePath );

                
END_METHOD

{attribute 'TcRpcEnable' := '1'}
METHOD load : RequestResults
  VAR_INPUT
    filePath : STRING;
  END_VAR
                  load := THIS^.processes.load.request( filePath := filePath );

                
END_METHOD

{attribute 'TcRpcEnable' := '1'}
METHOD activate : RequestResults
                  activate := THIS^.processes.activate.request();

                
END_METHOD

{attribute 'TcRpcEnable' := '1'}
METHOD _log : BOOL
  VAR_INPUT
    name : STRING;  (* Name of this function block instance *)
  END_VAR
  VAR_IN_OUT
    buffer : LogBuffer;  (* Buffer to write all logging to *)
  END_VAR
  VAR
    subBuffer : LogBuffer;  (* Temporary buffer to write logging by parts (sub-statemachines) to *)
  END_VAR
                  LOGGER(
    name := name,
    actualStatus := THIS^.actualStatus,
    previousStatus := THIS^.previousStatus,
    buffer := buffer,
    subBuffer := subBuffer,
    pHealthStatus := ADR(THIS^.statuses.healthStatus),
    pBusyStatus := ADR(THIS^.statuses.busyStatus));

                
END_METHOD
END_FUNCTION_BLOCK

FUNCTION_BLOCK SM_ModbusRTUBus
  VAR_INPUT
    {attribute 'OPC.UA.DA' := '1'}
    {attribute 'OPC.UA.DA.Access' := '1'}
    retries : INT := 3;  (* Number of retries for a succesfull process *)
    {attribute 'OPC.UA.DA' := '0'}
    isEnabled : BOOL;  (* Is control enabled? *)
  END_VAR
  VAR_OUTPUT
    {attribute 'OPC.UA.DA' := '1'}
    {attribute 'OPC.UA.DA.Access' := '1'}
    actualStatus : STRING;  (* Current status description *)
    previousStatus : STRING;  (* Previous status description *)
    statuses : ModbusRTUBusStatuses;  (* Statuses of the state machine *)
    processes : ModbusRTUBusProcesses;  (* Processes of the state machine *)
  END_VAR

            statuses.busyStatus( isBusy := processes.readCoil.statuses.busyStatus.busy OR (processes.writeCoil.statuses.busyStatus.busy OR (processes.readRegister.statuses.busyStatus.busy OR processes.writeRegister.statuses.busyStatus.busy)) );
processes.readCoil( isEnabled := isEnabled AND statuses.busyStatus.idle );
processes.writeCoil( isEnabled := isEnabled AND statuses.busyStatus.idle );
processes.readRegister( isEnabled := isEnabled AND statuses.busyStatus.idle );
processes.writeRegister( isEnabled := isEnabled AND statuses.busyStatus.idle );

          

{attribute 'TcRpcEnable' := '1'}
METHOD readCoil : RequestResults
  VAR_INPUT
    unitID : USINT;
    address : UINT;
  END_VAR
                  readCoil := THIS^.processes.readCoil.request(
    unitID := unitID,
    address := address);

                
END_METHOD

{attribute 'TcRpcEnable' := '1'}
METHOD writeCoil : RequestResults
  VAR_INPUT
    unitID : USINT;
    address : UINT;
    value : BOOL;
  END_VAR
                  writeCoil := THIS^.processes.writeCoil.request(
    unitID := unitID,
    address := address,
    value := value);

                
END_METHOD

{attribute 'TcRpcEnable' := '1'}
METHOD readRegister : RequestResults
  VAR_INPUT
    unitID : USINT;
    address : UINT;
  END_VAR
                  readRegister := THIS^.processes.readRegister.request(
    unitID := unitID,
    address := address);

                
END_METHOD

{attribute 'TcRpcEnable' := '1'}
METHOD writeRegister : RequestResults
  VAR_INPUT
    unitID : USINT;
    address : UINT;
    value : INT;
  END_VAR
                  writeRegister := THIS^.processes.writeRegister.request(
    unitID := unitID,
    address := address,
    value := value);

                
END_METHOD

{attribute 'TcRpcEnable' := '1'}
METHOD _log : BOOL
  VAR_INPUT
    name : STRING;  (* Name of this function block instance *)
  END_VAR
  VAR_IN_OUT
    buffer : LogBuffer;  (* Buffer to write all logging to *)
  END_VAR
  VAR
    subBuffer : LogBuffer;  (* Temporary buffer to write logging by parts (sub-statemachines) to *)
  END_VAR
                  LOGGER(
    name := name,
    actualStatus := THIS^.actualStatus,
    previousStatus := THIS^.previousStatus,
    buffer := buffer,
    subBuffer := subBuffer,
    pBusyStatus := ADR(THIS^.statuses.busyStatus));

                
END_METHOD
END_FUNCTION_BLOCK

FUNCTION_BLOCK Process EXTENDS BaseProcess
  VAR
    {attribute 'OPC.UA.DA' := '0'}
    testVar : BOOL;  (* At least 1 variable needed because subclass members of an empty class are not exposed by OPC UA (TwinCAT bug!) *)
  END_VAR

            IF do_request THEN
    do_request_result := request();
    do_request := FALSE;
END_IF;
SUPER^();

          

{attribute 'TcRpcEnable' := '1'}
METHOD start
                  THIS^.statuses.busyStatus( isBusy := TRUE );
THIS^.statuses.healthStatus( isGood := TRUE );

                
END_METHOD

{attribute 'TcRpcEnable' := '1'}
METHOD request : RequestResults
                  IF THIS^.statuses.enabledStatus.enabled THEN
    THIS^.start();
    request := RequestResults.ACCEPTED;
ELSE
    request := RequestResults.REJECTED;
END_IF;

                
END_METHOD
END_FUNCTION_BLOCK

FUNCTION_BLOCK McProcess EXTENDS BaseMcProcess
  VAR
    {attribute 'OPC.UA.DA' := '0'}
    testVar : BOOL;  (* At least 1 variable needed because subclass members of an empty class are not exposed by OPC UA (TwinCAT bug!) *)
  END_VAR

            IF do_request THEN
    do_request_result := request();
    do_request := FALSE;
END_IF;
SUPER^();

          

{attribute 'TcRpcEnable' := '1'}
METHOD start
                  THIS^.statuses.busyStatus( isBusy := TRUE );
THIS^.statuses.healthStatus( isGood := TRUE );

                
END_METHOD

{attribute 'TcRpcEnable' := '1'}
METHOD request : RequestResults
                  IF THIS^.statuses.enabledStatus.enabled THEN
    THIS^.start();
    request := RequestResults.ACCEPTED;
ELSE
    request := RequestResults.REJECTED;
END_IF;

                
END_METHOD
END_FUNCTION_BLOCK

FUNCTION_BLOCK ChangeSetpointProcess EXTENDS BaseProcess
  VAR_INPUT
    {attribute 'OPC.UA.DA' := '1'}
    set : ChangeSetpointProcessArgs;  (* Arguments to be set, before writing do_request TRUE *)
  END_VAR
  VAR_OUTPUT
    {attribute 'OPC.UA.DA' := '1'}
    {attribute 'OPC.UA.DA.Access' := '1'}
    get : ChangeSetpointProcessArgs;  (* Arguments in use by the process, if do_request was accepted *)
  END_VAR

            IF do_request THEN
    do_request_result := request( setpoint := set.setpoint );
    do_request := FALSE;
END_IF;
SUPER^();

          

{attribute 'TcRpcEnable' := '1'}
METHOD start
  VAR_INPUT
    setpoint : LREAL;  (* New setpoint value *)
  END_VAR
                  THIS^.get.setpoint := setpoint;
THIS^.statuses.busyStatus( isBusy := TRUE );
THIS^.statuses.healthStatus( isGood := TRUE );

                
END_METHOD

{attribute 'TcRpcEnable' := '1'}
METHOD request : RequestResults
  VAR_INPUT
    setpoint : LREAL;  (* New setpoint value *)
  END_VAR
                  IF THIS^.statuses.enabledStatus.enabled THEN
    THIS^.start( setpoint := setpoint );
    request := RequestResults.ACCEPTED;
ELSE
    request := RequestResults.REJECTED;
END_IF;

                
END_METHOD
END_FUNCTION_BLOCK

FUNCTION_BLOCK McMoveAbsoluteProcess EXTENDS BaseMcProcess
  VAR_INPUT
    {attribute 'OPC.UA.DA' := '1'}
    set : McMoveAbsoluteProcessArgs;  (* Arguments to be set, before writing do_request TRUE *)
  END_VAR
  VAR_OUTPUT
    {attribute 'OPC.UA.DA' := '1'}
    {attribute 'OPC.UA.DA.Access' := '1'}
    get : McMoveAbsoluteProcessArgs;  (* Arguments in use by the process, if do_request was accepted *)
  END_VAR

            IF do_request THEN
    do_request_result := request(
    position := set.position,
    maxVelocity := set.maxVelocity);
    do_request := FALSE;
END_IF;
SUPER^();

          

